// Calculate percent of register usage
IF ( CurrentAcrUsageCount > 0)
THEN
  CurrentAcrUsagePercent :=  (DINT_TO_REAL(CurrentAcrUsageCount) / DINT_TO_REAL(RegisterSize)) * 100.0;
ELSE
  CurrentAcrUsagePercent := 0.0;
END_IF

// build rising edge for arc usage over 80% 
WarningAcrUsage( CLK := CurrentAcrUsagePercent > RobotLibraryParameter.ACR_USAGE_WARNING_LIMIT );

IF ( WarningAcrUsage.Q )
THEN
  // Create log entry
  CreateLogMessagePara4( Timestamp   := SystemTime,
                         MessageType := MessageType.CMD,
                         Severity    := Severity.WARNING,
                         MessageCode := 0,
                         MessageText := 'ACR Register usage has reached the warning limit ({1}): {2}/{3} = {4}%',
                         Para1       :=  REAL_TO_STRING(RobotLibraryParameter.ACR_USAGE_WARNING_LIMIT),
                         Para2       :=  DINT_TO_STRING(CurrentAcrUsageCount),
                         Para3       :=  DINT_TO_STRING(RegisterSize),
                         Para4       :=  REAL_TO_STRING(CurrentAcrUsagePercent));  
END_IF
                
END_METHOD

METHOD PUBLIC OnOnlineChange : DINT
VAR_INPUT
  /// unique ID 
  UniqueID     : UDINT;
  /// Pointer to the corresponding command-FB to enable a callback mechanism
  pCommandFB   : POINTER TO RobotLibraryBaseFB;
END_VAR

VAR
  /// internal index for loops
 _regIdx : DINT;
END_VAR
                  OnOnlineChange := -1;

// Check command FB pointer is valid ?
IF ( pCommandFB <> RobotLibraryConstants.NULL_POINTER)
THEN
  FOR _regIdx := 1 TO RegisterSize
  DO
    // check unique ID found ?
    IF ( Register[_regIdx].UniqueID = UniqueID ) 
    THEN  
      // update pointer to command FB
      Register[_regIdx].pCommandFB := pCommandFB;
      // Return result OK
      OnOnlineChange := RobotLibraryConstants.OK;
      EXIT;
    END_IF
  END_FOR
END_IF
                
END_METHOD

METHOD PUBLIC RemoveCmd : DINT
VAR_INPUT
 /// unique ID
 UniqueID : UDINT;  
END_VAR

VAR
  /// internal index
 _regIdx : DINT;
  /// internal command type 
 _cmdType : CmdType;
END_VAR
                  RemoveCmd := RobotLibraryConstants.HAS_ERROR;


IF (UniqueID = 0)
THEN
  UniqueID := UniqueID;
END_IF

FOR _regIdx := 1 TO RegisterSize
DO
  // check unique ID found and not yet sended ?
  IF (( Register[_regIdx].UniqueID                  = UniqueID                        ) AND
      ( Register[_regIdx].Command[ACTIVE_CMD].State < BufferStateCmd.UPDATE_AVAILABLE ))       
  THEN
    // Get CmdType from payload
    SysDepMemCpy( pDest := ADR(_cmdType), pSrc := ADR(Register[_regIdx].Command[ACTIVE_CMD].Payload), DataLen := SIZEOF(_cmdType));
    // delete register entry
    SysDepMemSet(pDest := ADR(Register[_regIdx]), Value := 0 , DataLen := SIZEOF(Register[_regIdx]));
    // decrement current used register counter
    CurrentAcrUsageCount := CurrentAcrUsageCount - 1;
    // Command successfull removed
    RemoveCmd := RobotLibraryConstants.OK;    
    
    
    // Create log entry
    CreateLogMessagePara2 (  Timestamp   := SystemTime,
                             MessageType := MessageType.CMD,
                             Severity    := Severity.INFO,
                             MessageCode := 0,
                             MessageText := 'ACR-ID [{1}]: Removed CmdType <{2}>',
                             Para1       :=  DINT_TO_STRING(_regIdx),                 
                             Para2       :=  CMD_TYPE_TO_STRING(SwapUint(_cmdType)));
    EXIT;
  END_IF
END_FOR
                
END_METHOD

METHOD PUBLIC Reset
                  SysDepMemSet( ADR(Register), 0, SIZEOF(Register));              

CurrentAcrUsageCount   := 0;
CurrentAcrUsagePercent := 0.0;


// Create log entry
CreateLogMessagePara1 ( Timestamp   := SystemTime,
                        MessageType := MessageType.CMD,
                        Severity    := Severity.INFO,
                        MessageCode := 0,
                        MessageText := 'ACR Registers has been reset and all entries deleted by Reset method call',
                        Para1       :=  '');                          

                
END_METHOD

METHOD PRIVATE UpdateExecutionOrderList
VAR
  /// temporary Active Command Register entry
  TmpRegisterEntry : AxesGroupAcyclicAcrEntry;
  /// temporary index
  TmpIndex         : DINT;
  /// internal index
  i                : DINT;  
  /// internal index
  j                : DINT;  
END_VAR
                  // Reset temporary register
SysDepMemSet(pDest := ADR(TmpRegister)       , Value := 0, DataLen := SIZEOF(TmpRegister));
// Reset Execution Order List
SysDepMemSet(pDest := ADR(ExecutionOrderList), Value := 0, DataLen := SIZEOF(ExecutionOrderList));
// pre-set temporary register index 
j := 1;

FOR i := 1 TO RegisterSize
DO
  // add only entries which are not in status free and where datas must be processed
  IF (( Register[i].State                      > ActiveCommandRegisterState.IS_FREE ) AND
      ( Register[i].Command[ACTIVE_CMD].State <> BufferStateCmd.EMPTY               ) AND
      ( Register[i].Command[ACTIVE_CMD].State <> BufferStateCmd.PROCESSED           ))
  THEN
    // copy register entry 
    TmpRegister[j] := Register[i];
    // store index of the entry from the ACR
    ExecutionOrderList[j] := i;
    // inc temporar register index
    j := j + 1; 
  END_IF
END_FOR  

// Bubble Sort to sort the priorities from the active command register
FOR i := 1 TO RegisterSize
DO
  FOR j := 1 TO RegisterSize - 1
  DO 
    // check list entry is not empty ? 
    IF (( TmpRegister[i  ].State = ActiveCommandRegisterState.IS_FREE ) OR
        ( TmpRegister[j+1].State = ActiveCommandRegisterState.IS_FREE ))
    THEN
      EXIT; 
    END_IF  

    IF (( TmpRegister[j].Command[ACTIVE_CMD].Payload[PRIORITY_IDX] AND PRIORITY_BIT_MASK ) > ( TmpRegister[j+1].Command[ACTIVE_CMD].Payload[PRIORITY_IDX] AND PRIORITY_BIT_MASK ))
    THEN    
      // swap position of register entry  
      TmpRegisterEntry := TmpRegister[j];         
      TmpRegister[j]   := TmpRegister[j+1];
      TmpRegister[j+1] := TmpRegisterEntry;
      
      // swap position of index in the Execution Order List  
      TmpIndex                := ExecutionOrderList[j];
      ExecutionOrderList[j]   := ExecutionOrderList[j+1];
      ExecutionOrderList[j+1] := TmpIndex;
    END_IF
  END_FOR 
END_FOR

// Bubble Sort to sort the Timestamp from the pre-sorted active command register
FOR i := 1 TO RegisterSize
DO
  FOR j := 1 TO RegisterSize - 1
  DO    
    // check list entry is not empty ? 
    IF (( TmpRegister[i  ].State = ActiveCommandRegisterState.IS_FREE ) OR
        ( TmpRegister[j+1].State = ActiveCommandRegisterState.IS_FREE ))
    THEN
      EXIT; 
    END_IF  

       // Priority is higher
    IF (( TmpRegister[j].Command[ACTIVE_CMD].Payload[PRIORITY_IDX] AND PRIORITY_BIT_MASK ) >= ( TmpRegister[j+1].Command[ACTIVE_CMD].Payload[PRIORITY_IDX] AND PRIORITY_BIT_MASK )) AND
       // Date is greater 
       (( TmpRegister[j].Command[ACTIVE_CMD].Timestamp.SystemDate                          >    TmpRegister[j+1].Command[ACTIVE_CMD].Timestamp.SystemDate                         ) OR 
       // Date is the same, but Time is greater
       (( TmpRegister[j].Command[ACTIVE_CMD].Timestamp.SystemDate                          =    TmpRegister[j+1].Command[ACTIVE_CMD].Timestamp.SystemDate                         ) AND 
        ( TmpRegister[j].Command[ACTIVE_CMD].Timestamp.SystemTime                          >    TmpRegister[j+1].Command[ACTIVE_CMD].Timestamp.SystemTime                         )))
    THEN    
      // swap position of register entry  
      TmpRegisterEntry := TmpRegister[j];         
      TmpRegister[j]   := TmpRegister[j+1];
      TmpRegister[j+1] := TmpRegisterEntry;
      
      // swap position of index in the Execution Order List  
      TmpIndex                := ExecutionOrderList[j];
      ExecutionOrderList[j]   := ExecutionOrderList[j+1];
      ExecutionOrderList[j+1] := TmpIndex;
    END_IF
  END_FOR 
END_FOR
                
END_METHOD

PROPERTY PUBLIC NotifyParameterChanged : UDINT
SET
VAR
  /// internal register index
 _regIdx  : DINT;
  /// internal command type
 _cmdType : CmdType;
END_VAR
                    FOR _regIdx := 1 TO RobotLibraryParameter.ACTIVE_CMD_REGISTER_ENTRIES_MAX
DO
  // check unique ID found ?
  IF ( Register[_regIdx].UniqueID = NotifyParameterChanged )
  THEN  
    IF (( Register[_regIdx].Command[ACTIVE_CMD].State <> BufferStateCmd.SENDING   ) AND
        ( Register[_regIdx].Command[ACTIVE_CMD].State <> BufferStateCmd.PROCESSED ))
    THEN
      // Check pointer is valid ? 
      IF ( Register[_regIdx].pCommandFB <> RobotLibraryConstants.NULL_POINTER )
      THEN
        // add to send register
        Register[_regIdx].Command[ACTIVE_CMD].Timestamp  := SystemTime;
        Register[_regIdx].Command[ACTIVE_CMD].State      := BufferStateCmd.UPDATE_AVAILABLE;
        Register[_regIdx].Command[ACTIVE_CMD].Payload    := Register[_regIdx].pCommandFB^.CommandData.Payload;
        Register[_regIdx].Command[ACTIVE_CMD].PayloadLen := Register[_regIdx].pCommandFB^.CommandData.PayloadLen;

        // get command type from payload
       _cmdType := CombineBytesToUint(HiByte := Register[_regIdx].pCommandFB^.CommandData.Payload[0],
                                      LoByte := Register[_regIdx].pCommandFB^.CommandData.Payload[1]);
        
        // Create log entry
        CreateLogMessagePara2 ( Timestamp   := SystemTime,
                                MessageType := MessageType.CMD,
                                Severity    := Severity.INFO,
                                MessageCode := 0,
                                MessageText := 'ACR-ID [{1}]: Updated Cmd-Parameter of CmdType <{2}> -> written to ACTIVE_CMD Index',
                                Para1       :=  DINT_TO_STRING(_regIdx),
                                Para2       :=  CMD_TYPE_TO_STRING(_cmdType));
      END_IF
    ELSE
      // Check pointer is valid ? 
      IF ( Register[_regIdx].pCommandFB <> RobotLibraryConstants.NULL_POINTER )
      THEN
        // add to buffer register
        Register[_regIdx].Command[BUFFER_CMD].Timestamp  := SystemTime;
        Register[_regIdx].Command[BUFFER_CMD].State      := BufferStateCmd.UPDATE_AVAILABLE;
        Register[_regIdx].Command[BUFFER_CMD].Payload    := Register[_regIdx].pCommandFB^.CommandData.Payload;
        Register[_regIdx].Command[BUFFER_CMD].PayloadLen := Register[_regIdx].pCommandFB^.CommandData.PayloadLen;

        // get command type from payload
       _cmdType := CombineBytesToUint(HiByte := Register[_regIdx].pCommandFB^.CommandData.Payload[0],
                                      LoByte := Register[_regIdx].pCommandFB^.CommandData.Payload[1]);
        
        // Create log entry
        CreateLogMessagePara2 ( Timestamp   := SystemTime,
                                MessageType := MessageType.CMD,
                                Severity    := Severity.INFO,
                                MessageCode := 0,
                                MessageText := 'ACR-ID [{1}]: Updated Cmd-Parameter of CmdType <{2}> -> written to BUFFER_CMD Index',
                                Para1       :=  DINT_TO_STRING(_regIdx),
                                Para2       :=  CMD_TYPE_TO_STRING(_cmdType));
      END_IF
    END_IF
    
    
  END_IF
END_FOR
                  
END_SET
END_PROPERTY
END_FUNCTION_BLOCK

/// Abort triggering of Position, measuring input
FUNCTION_BLOCK MC_AbortMeasuringInputFB EXTENDS RobotLibraryBaseExecuteFB
// ------------------------------------------------------------------------- 
//  SRCI Robot Library                                                
// ------------------------------------------------------------------------- 
//                                                                           
//  Object:      AbortMeasuringInputFB                                       
//  Author:      Thorsten Brach                                                
//  Date:        2024-06-01
//
//  Description:                                              
//   
//                                                                           
//  Copyright: 
//    (C) 2024 Thorsten Brach. All rights reserved                                                                                                                                            
//             Licensed under the MIT License.
//                                                                           
//  Disclaimer:                                                                           
//    This project is provided without any guarantee and can be used for   
//    private and commercial purposes. Any use is at the user’s 
//    own risk and responsibility.
//
// -------------------------------------------------------------------------
VAR_INPUT
  /// Command parameter 
  ParCmd          : AbortMeasuringInputParCmd;      
END_VAR
VAR_OUTPUT
  /// Command is transferred and confirmed by the RC
  CommandBuffered : BOOL;  
  /// Command output 
  OutCmd          : AbortMeasuringInputOutCmd;          
END_VAR
VAR
  /// internal copy of command parameter 
 _parCmd          : AbortMeasuringInputParCmd;
  /// command data to send
 _command         : AbortMeasuringInputSendData;
  /// response data received
 _response        : AbortMeasuringInputRecvData;      
END_VAR

            SUPER^(AxesGroup := AxesGroup);
          

METHOD INTERNAL CheckAddParameter : BOOL
VAR_INPUT
  /// Payload pointer
  PayloadPtr : UDINT;
END_VAR
VAR
  /// Payload as byte array
  Payload    : ARRAY [1..SIZEOF(_command)] OF BYTE;
  /// Null Byte array 
  Null       : ARRAY [1..SIZEOF(_command)] OF BYTE;
  /// Data length to compare
  DataLen    : UDINT;
END_VAR
                  // Payload pointer must be decreased by one byte, because ADR(Payload) is already one byte !
PayloadPtr := LIMIT (0, PayloadPtr - 1, SIZEOF(Payload) -1);
// Convert command struct to payload array
SysDepMemCpy( pDest := ADR(Payload), pSrc := ADR(_command), DataLen := SIZEOF(_command));
// Calculate the data length to compare - at least one byte must be compared !
DataLen := LIMIT(1, SIZEOF(Payload) - PayloadPtr, SIZEOF(Payload)); 
// Compare Payload-Array with Null-Byte-Array
CheckAddParameter := SysDepMemCmp( pData1 := ADR(Payload) + PayloadPtr , pData2 := ADR(Null), DataLen := DataLen) <>  RobotLibraryConstants.OK ;
                
END_METHOD

METHOD PROTECTED CheckFunctionSupported : BOOL
VAR_IN_OUT
  /// Robot assignment of function
  AxesGroup : AxesGroup; 
END_VAR
                  CheckFunctionSupported := AxesGroup.State.RobotData.RCSupportedFunctions.AbortMeasuringInput;

IF ( NOT CheckFunctionSupported )
THEN
  // call base implementation for set error and create log entry
  SUPER^.CheckFunctionSupported(AxesGroup := AxesGroup);
END_IF
                
END_METHOD

METHOD PROTECTED CheckParameterChanged : BOOL
VAR_IN_OUT
  /// Robot assignment of function
  AxesGroup    : AxesGroup; 
END_VAR
                  // Check ParCmd Size is > 0, because MemCmp does not work correctly with size = 0
IF (SIZEOF(ParCmd) = 0) OR (_stepCmd = 0)
THEN 
  RETURN;
END_IF

// compare memory 
_parameterChanged := ( SysDepMemCmp(pData1 := ADR(ParCmd), pData2 := ADR(_parCmd), DataLen := SIZEOF(ParCmd)) <> RobotLibraryConstants.OK );

// check parameter valid ?
_parameterValid   := CheckParameterValid( AxesGroup := AxesGroup );

IF ((  _parameterChanged        )  AND 
    (  _parameterValid          )) OR
    (  _parameterUpdateInternal )  
THEN  
  // Create log entry for parameter changed event
  CreateLogMessagePara1 ( Timestamp   := AxesGroup.State.SystemTime,
                          MessageType := MessageType.CMD,
                          Severity    := Severity.DEBUG,
                          MessageCode := 0,
                          MessageText := 'NotifyParameterChanged Event {1}',
                          Para1       :=  '' );

  // reset internal flag for send parameter update
 _parameterUpdateInternal := FALSE;
  // update internal copy of parameters 
 _parCmd := ParCmd;
  // inc parameter sequence
 _command.ParSeq := _command.ParSeq + 1;
  // update command data  
  CommandData := CreateCommandPayload(AxesGroup := AxesGroup); // ( Access via reference to rCommandFB in ACR )
  // notify active command register 
  AxesGroup.Acyclic.ActiveCommandRegister.NotifyParameterChanged := _uniqueID;
END_IF
                
END_METHOD

METHOD PROTECTED CheckParameterValid : BOOL
VAR_IN_OUT
  /// Robot assignment of function
  AxesGroup : AxesGroup; 
END_VAR
                  CheckParameterValid := TRUE;


// Check ParCmd.MeasuringID valid ? 
IF ( ParCmd.MeasuringID < 0 )
THEN
  // Parameter not valid
  CheckParameterValid := FALSE;
  // Set error
  SetError( ErrorID := RobotLibraryErrorIdEnum.ERR_INVALID_PAR_CMD, Overwrite := TRUE ); 
  // Create log entry
  CreateLogMessagePara1 ( Timestamp   := AxesGroup.State.SystemTime,
                          MessageType := MessageType.CMD,
                          Severity    := Severity.ERROR,
                          MessageCode := ErrorID,
                          MessageText := 'Invalid Parameter ParCmd.MeasuringID = {1}',
                          Para1       := UINT_TO_STRING(ParCmd.MeasuringID));
  RETURN;                          
END_IF
                
END_METHOD

METHOD INTERNAL CreateCommandPayload : RobotLibraryCommandDataFB
VAR_IN_OUT
  /// Robot assignment of function
  AxesGroup : AxesGroup; 
END_VAR
VAR
  /// Parameter count
 _parameterCnt : DINT;
END_VAR
// Table 6-571: Sent CMD payload (PLC to RC) of "AbortMeasuringInput"
// --------------------------
// Header
// --------------------------
// Byte 000 : UINT  - Type HB     
// Byte 001 :       - Type LB    
// Byte 002 : USINT - Reserve | ExecutionMode
// Byte 003 : USINT - ParSeq  | Priority
// --------------------------
// Datablock
// --------------------------
// Byte 004 : UINT       - MeasuringID LW HB
// Byte 005 :            - MeasuringID LW LB
                  // set command parameter 
_command.CmdTyp      :=  CmdType.AbortMeasuringInput;
_command.ExecMode    :=  ExecMode;
_command.ParSeq      := _command.ParSeq;
_command.Priority    :=  Priority;
                     
_command.MeasuringID := parCmd.MeasuringID;

// copy command data to header
_cmdHeader := _command;
// call base implementation to copy header to payload buffer
CreateCommandPayload := SUPER^.CreateCommandPayload(AxesGroup := AxesGroup);


// Check parameter must be added ? 
IF ( CheckAddParameter(CreateCommandPayload.PayloadPtr))
THEN
  // add command.MeasuringID
  CreateCommandPayload.AddUint(_command.MeasuringID);
  // inc parameter counter
 _parameterCnt := _parameterCnt + 1;  
END_IF


// Create logging
CreateCommandPayloadLog(AxesGroup := AxesGroup, ParameterCnt := _parameterCnt);
                
END_METHOD

METHOD INTERNAL CreateCommandPayloadLog
VAR_IN_OUT
  /// Robot assignment of function
  AxesGroup : AxesGroup; 
END_VAR
VAR_INPUT
  /// Parameter count
  ParameterCnt : DINT;
END_VAR
                  // Create log entry for Parameter start
CreateLogMessagePara1 ( Timestamp   := AxesGroup.State.SystemTime,
                        MessageType := MessageType.CMD,
                        Severity    := Severity.DEBUG,
                        MessageCode := 0,
                        MessageText := 'Create command payload with {1} parameter(s) :',
                        Para1       := DINT_TO_STRING(ParameterCnt));
  

// Return if no parameter is remaining...
IF ( ParameterCnt = 0 ) THEN RETURN; END_IF
// dec remaining parameter(s)                        
ParameterCnt := ParameterCnt - 1;
// Create log entry for MeasuringID
CreateLogMessagePara1 ( Timestamp   := AxesGroup.State.SystemTime,
                        MessageType := MessageType.CMD,
                        Severity    := Severity.DEBUG,
                        MessageCode := 0,
                        MessageText := 'Command.MeasuringID = {1}',
                        Para1       :=  UINT_TO_STRING(_command.MeasuringID));

                
END_METHOD

METHOD FB_init : BOOL
VAR_INPUT
  /// if TRUE, the retain variables are initialized (warm start / cold start)
  bInitRetains : BOOL; 
  /// if TRUE, the instance afterwards gets moved into the copy code (online change)
  bInCopyCode  : BOOL;  
END_VAR
                  MyType := 'MC_AbortMeasuringInputFB';

ExecMode := ExecutionMode.PARALLEL;
Priority := PriorityLevel.NORMAL;
                
END_METHOD

METHOD PROTECTED OnExecRun : DINT
VAR_IN_OUT
  /// Robot assignment of function
  AxesGroup : AxesGroup; 
END_VAR
                  // call base implementation
SUPER^.OnExecRun(AxesGroup := AxesGroup);

CASE _stepCmd OF
  
  00:  IF ( _execute_R.Q ) AND ( NOT Error)
       THEN
         // Check function is supported and parameter are valid ?
         IF (( CheckFunctionSupported( AxesGroup := AxesGroup )) AND
             ( CheckParameterValid   ( AxesGroup := AxesGroup )))      
         THEN
           // set busy flag
           Busy := TRUE;
           // Reset command outputs
           SysDepMemSet(pDest := ADR(OutCmd), Value := 0, DataLen := SIZEOF(OutCmd));         
           // apply command parameter
          _parCmd := ParCmd;
           // init parameter sequence
          _command.ParSeq := 1;
           // create command data
           CommandData := CreateCommandPayload(AxesGroup := AxesGroup);
           // Add command to active command register
          _uniqueID := AxesGroup.Acyclic.ActiveCommandRegister.AddCmd( pCommandFB := ADR(THIS^ ));     
           // set timeout
           SetTimeout(PT := _timeoutCmd, rTimer := _timerCmd);
           // inc step counter
          _stepCmd := _stepCmd + 1;
         END_IF 
       END_IF


  01:  // Wait for responce received
       IF ( _responseReceived )
       THEN
         // reset response received flag
        _responseReceived := FALSE;
         // update state flags
         OnUpdateStateFlags(_response.State);
         // update state flags
         OnApplyOutCmd(_response.State);
                
         // Done, Aborted or Error ?
         IF (_response.State >= CmdMessageState.DONE )
         THEN
           // set timeout
           SetTimeout(PT := _timeoutCmd, rTimer := _timerCmd);
           // inc step counter
          _stepCmd := _stepCmd + 1; 
         END_IF
       END_IF


  02: IF ( NOT Execute)
      THEN
        Reset();
      END_IF     
ELSE
  // invalid step
  SetError( ErrorID := RobotLibraryErrorIdEnum.ERR_INVALID_STEP, Overwrite := TRUE );
END_CASE


// Reset FB
IF ( NOT Execute )
THEN
  Reset();
END_IF
                
END_METHOD

METHOD PROTECTED OnUpdateStateFlags
VAR_INPUT
  /// Command message state
  State : CmdMessageState;
END_VAR
                  // Reset State flags
Done:= FALSE;

CASE State OF

  // No operation or process is active
  CmdMessageState.EMPTY               :;
  // Created but not yet started
  CmdMessageState.CREATED             :;
  // Buffered and awaiting execution
  CmdMessageState.BUFFERED            : CommandBuffered := TRUE;
  // Buffered in planner for future execution
  CmdMessageState.BUFFERED_IN_PLANNER : CommandBuffered := TRUE;
  // Currently active and in progress
  CmdMessageState.ACTIVE              :;
  // Interrupted and awaiting continuation
  CmdMessageState.INTERRUPTED         :;
  // Requested for abort
  CmdMessageState.ABORT_REQUEST       :;
  // Successfully completed
  CmdMessageState.DONE                : Done  := TRUE;
                                        Busy  := FALSE;
  // Aborted before completion
  CmdMessageState.ABORTED             : Busy  := FALSE;
  // Encountered an error during execution
  CmdMessageState.ERROR               : Error := TRUE;
                                        Busy  := FALSE;
END_CASE
                
END_METHOD

METHOD INTERNAL ParseResponsePayload : DINT
VAR_INPUT
  /// Response data
  ResponseData : RobotLibraryResponseDataFB;
  /// Timestamp
  Timestamp    : SystemTime;  
END_VAR
VAR
  /// Parameter count
 _parameterCnt : DINT;
END_VAR
// Table 6-572: Received CMD payload (RC to PLC) of "AbortMeasuringInput"
// --------------------------
// Header
// --------------------------
// Byte 00 : USINT - ParSeq | State     
// Byte 01 : SINT  - AlarmMessageSeverity    
// Byte 02 : UINT  - AlarmMessageCode HB
// Byte 03 :       - AlarmMessageCode LB
                  // call base implementation to parse the header from payload buffer
ResponseData.PayloadPtr := SUPER^.ParseResponsePayload(ResponseData := ResponseData, Timestamp := Timestamp);

// copy parsed header to response
_response.ParSeq               := _rspHeader.ParSeq;
_response.State                := _rspHeader.State;
_response.AlarmMessageSeverity := _rspHeader.AlarmMessageSeverity;
_response.AlarmMessageCode     := _rspHeader.AlarmMessageCode;

// Create logging
ParseResponsePayloadLog(ResponseData := ResponseData, Timestamp := Timestamp, ParameterCnt := _parameterCnt);
                
END_METHOD

METHOD INTERNAL ParseResponsePayloadLog
VAR_INPUT
  /// Response data
  ResponseData : RobotLibraryResponseDataFB;
  /// Timestamp
  Timestamp    : SystemTime;  
  /// Parameter count
  ParameterCnt : DINT;
END_VAR
                  // Create log entry for Parameter start
CreateLogMessagePara1 ( Timestamp   := Timestamp,
                        MessageType := MessageType.CMD,
                        Severity    := Severity.DEBUG,
                        MessageCode := 0,
                        MessageText := '{1} parameter(s) to parse from the response data:',
                        Para1       := DINT_TO_STRING(ParameterCnt));
                        
// Return if no parameter is remaining...
IF ( ParameterCnt = 0 ) THEN RETURN; END_IF
// dec remaining parameter(s)                        
ParameterCnt := ParameterCnt - 1;
// Create log entry for no parameter 
CreateLogMessage      ( Timestamp   := Timestamp,
                        MessageType := MessageType.CMD,
                        Severity    := Severity.DEBUG,
                        MessageCode := 0,
                        MessageText := 'This command has no parameter to parse...');
                
END_METHOD

METHOD PROTECTED Reset : DINT
VAR_INPUT
END_VAR
                  Reset := SUPER^.Reset();

Done            := FALSE;
Busy            := FALSE;
CommandBuffered := FALSE;
                
END_METHOD
END_FUNCTION_BLOCK

/// Cancel currently active move command and continue with the next buffered command
FUNCTION_BLOCK MC_ActivateNextCommandFB EXTENDS RobotLibraryBaseExecuteFB
// ------------------------------------------------------------------------- 
//  SRCI Robot Library                                                
// ------------------------------------------------------------------------- 
//                                                                           
//  Object:      ActivateNextCommandFB                                       
//  Author:      Thorsten Brach                                                
//  Date:        2024-06-01
//
//  Description:                                              
//   
//                                                                           
//  Copyright: 
//    (C) 2024 Thorsten Brach. All rights reserved                                                                                                                                            
//             Licensed under the MIT License.
//                                                                           
//  Disclaimer:                                                                           
//    This project is provided without any guarantee and can be used for   
//    private and commercial purposes. Any use is at the user’s 
//    own risk and responsibility.
//
// -------------------------------------------------------------------------
VAR_INPUT
  /// Command parameter 
  ParCmd          : ActivateNextCommandParCmd;
  /// Processing mode
  ProcessingMode  : ProcessingMode;  
END_VAR
VAR_OUTPUT
  /// Command is transferred and confirmed by the RC
  CommandBuffered : BOOL;
  /// command results
  OutCmd          : ActivateNextCommandOutCmd;
END_VAR

VAR
  /// internal copy of command parameter 
 _parCmd          : ActivateNextCommandParCmd;
  /// command data to send
 _command         : ActivateNextCommandSendData;
  /// response data received
 _response        : ActivateNextCommandRecvData;   
  /// Trigger related EmitterID
 _emitterID       : ARRAY[0..3] OF SINT;
END_VAR

            SUPER^(AxesGroup := AxesGroup);
          

METHOD INTERNAL CheckAddParameter : BOOL
VAR_INPUT
  /// Payload pointer
  PayloadPtr : UDINT;
END_VAR
VAR
  /// Payload as byte array
  Payload    : ARRAY [1..SIZEOF(_command)] OF BYTE;
  /// Null Byte array 
  Null       : ARRAY [1..SIZEOF(_command)] OF BYTE;
  /// Data length to compare
  DataLen    : UDINT;
END_VAR
                  // Payload pointer must be decreased by one byte, because ADR(Payload) is already one byte !
PayloadPtr := LIMIT (0, PayloadPtr - 1, SIZEOF(Payload) -1);
// Convert command struct to payload array
SysDepMemCpy( pDest := ADR(Payload), pSrc := ADR(_command), DataLen := SIZEOF(_command));
// Calculate the data length to compare - at least one byte must be compared !
DataLen := LIMIT(1, SIZEOF(Payload) - PayloadPtr, SIZEOF(Payload)); 
// Compare Payload-Array with Null-Byte-Array
CheckAddParameter := SysDepMemCmp( pData1 := ADR(Payload) + PayloadPtr , pData2 := ADR(Null), DataLen := DataLen) <>  RobotLibraryConstants.OK ;
                
END_METHOD

METHOD PROTECTED CheckFunctionSupported : BOOL
VAR_IN_OUT
  /// Robot assignment of function
  AxesGroup : AxesGroup; 
END_VAR
                  CheckFunctionSupported := AxesGroup.State.RobotData.RCSupportedFunctions.ActivateNextCommand;

IF ( NOT CheckFunctionSupported )
THEN
  // call base implementation for set error and create log entry
  SUPER^.CheckFunctionSupported(AxesGroup := AxesGroup);
END_IF
                
END_METHOD

METHOD PROTECTED CheckParameterChanged : BOOL
VAR_IN_OUT
  /// Robot assignment of function
  AxesGroup    : AxesGroup; 
END_VAR
                  // Check ParCmd Size is > 0, because MemCmp does not work correctly with size = 0
IF (SIZEOF(ParCmd) = 0) OR (_stepCmd = 0)
THEN 
  RETURN;
END_IF

// compare memory 
_parameterChanged := ( SysDepMemCmp(pData1 := ADR(ParCmd), pData2 := ADR(_parCmd), DataLen := SIZEOF(ParCmd)) <> RobotLibraryConstants.OK );

// check parameter valid ?
_parameterValid   := CheckParameterValid( AxesGroup := AxesGroup );

IF ((  _parameterChanged        )  AND 
    (  _parameterValid          )) OR
    (  _parameterUpdateInternal )  
THEN  
  // Create log entry for parameter changed event
  CreateLogMessagePara1 ( Timestamp   := AxesGroup.State.SystemTime,
                          MessageType := MessageType.CMD,
                          Severity    := Severity.DEBUG,
                          MessageCode := 0,
                          MessageText := 'NotifyParameterChanged Event {1}',
                          Para1       :=  '' );

  // reset internal flag for send parameter update
 _parameterUpdateInternal := FALSE;
  // update internal copy of parameters 
 _parCmd := ParCmd;
  // inc parameter sequence
 _command.ParSeq := _command.ParSeq + 1;
  // update command data  
  CommandData := CreateCommandPayload(AxesGroup := AxesGroup); // ( Access via reference to rCommandFB in ACR )
  // notify active command register 
  AxesGroup.Acyclic.ActiveCommandRegister.NotifyParameterChanged := _uniqueID;  
END_IF
                
END_METHOD

METHOD PROTECTED CheckParameterValid : BOOL
VAR_IN_OUT
  /// Robot assignment of function
  AxesGroup : AxesGroup; 
END_VAR
                  CheckParameterValid := TRUE;

// Check ParCmd.ProcessingMode defined ? 
IF (( ProcessingMode < ProcessingModeEnum.BUFFERED         ) AND
    ( ProcessingMode > ProcessingModeEnum.TRIGGER_MULTIPLE ))
THEN
  // Parameter not valid
  CheckParameterValid := FALSE;
  // Set error
  SetError( ErrorID := RobotLibraryErrorIdEnum.ERR_PROCESSINGMODE_NOT_DEFINED, Overwrite := TRUE );
  // Create log entry
  CreateLogMessagePara1 ( Timestamp   := AxesGroup.State.SystemTime,
                          MessageType := MessageType.CMD,
                          Severity    := Severity.ERROR,
                          MessageCode := ErrorID,
                          MessageText := 'Invalid Parameter ParCmd.ProcessingMode = {1}',
                          Para1       := PROCESSING_MODE_TO_STRING(ProcessingMode));
  RETURN;                          
END_IF


// Check ParCmd.ProcessingMode valid ? 
IF (( ProcessingMode <> ProcessingModeEnum.PARALLEL         ) AND
    ( ProcessingMode <> ProcessingModeEnum.DEACTIVATE       ) AND
    ( ProcessingMode <> ProcessingModeEnum.TRIGGER_ONCE     ) AND
    ( ProcessingMode <> ProcessingModeEnum.TRIGGER_MULTIPLE ))
THEN
  // Parameter not valid
  CheckParameterValid := FALSE;
  // Set error
  SetError( ErrorID := RobotLibraryErrorIdEnum.ERR_PROCESSINGMODE_NOT_ALLOWED, Overwrite := TRUE );
  // Create log entry
  CreateLogMessagePara1 ( Timestamp   := AxesGroup.State.SystemTime,
                          MessageType := MessageType.CMD,
                          Severity    := Severity.ERROR,
                          MessageCode := ErrorID,
                          MessageText := 'Invalid Parameter ParCmd.ProcessingMode = {1}',
                          Para1       := PROCESSING_MODE_TO_STRING(ProcessingMode));
  RETURN;                          
END_IF


// Check ParCmd.ListenerID valid ? 
IF (( ParCmd.ListenerID <   0 ) OR 
    ( ParCmd.ListenerID > 127 ))
THEN
  // Parameter not valid
  CheckParameterValid := FALSE;
  // Set error
  SetError( ErrorID := RobotLibraryErrorIdEnum.ERR_LISTENERID_MUST_BE_POSITIVE, Overwrite := TRUE );
  // Create log entry
  CreateLogMessagePara1 ( Timestamp   := AxesGroup.State.SystemTime,
                          MessageType := MessageType.CMD,
                          Severity    := Severity.ERROR,
                          MessageCode := ErrorID,
                          MessageText := 'Invalid Parameter ParCmd.ListenerID = {1}',
                          Para1       := SINT_TO_STRING(ParCmd.ListenerID));                            
  RETURN;
END_IF


                
END_METHOD

METHOD INTERNAL CreateCommandPayload : RobotLibraryCommandDataFB
VAR_IN_OUT
  /// Robot assignment of function
  AxesGroup : AxesGroup; 
END_VAR
VAR
  /// Parameter count
 _parameterCnt : DINT;
END_VAR
// Table 6-662: Sent CMD payload (PLC to RC) of "ActivateNextCommand"
// --------------------------
// Header
// --------------------------
// Byte 00 : UINT  - Type HB     
// Byte 01 :       - Type LB    
// Byte 02 : USINT - Reserve | ExecutionMode
// Byte 03 : USINT - ParSeq  | Priority
// --------------------------
// Datablock
// --------------------------
// Byte 04 : SINT - EmitterID[0]
// Byte 05 : SINT - EmitterID[1]
// Byte 06 : SINT - EmitterID[2]   
// Byte 07 : SINT - EmitterID[3]
// Byte 08 : SINT - ListenerID
// Byte 09 : BYTE - Reserve
// --------------------------
                  // set command parameter 
_command.CmdTyp     :=  CmdType.ActivateNextCommand;
_command.ExecMode   :=  ExecMode;
_command.ParSeq     := _command.ParSeq;
_command.Priority   :=  Priority;
_command.ListenerID := _parCmd.ListenerID;


// copy command data to header
_cmdHeader := _command;
// call base implementation to copy header to payload buffer
CreateCommandPayload := SUPER^.CreateCommandPayload(AxesGroup := AxesGroup);


// Check parameter must be added ? 
IF ( CheckAddParameter(CreateCommandPayload.PayloadPtr))
THEN
  // add command.EmitterID[0]
  CreateCommandPayload.AddSint(_command.EmitterID[0]);
  // inc parameter counter
 _parameterCnt := _parameterCnt + 1;  
END_IF


// Check parameter must be added ? 
IF ( CheckAddParameter(CreateCommandPayload.PayloadPtr))
THEN
  // add command.EmitterID[1]
  CreateCommandPayload.AddSint(_command.EmitterID[1]);
  // inc parameter counter
 _parameterCnt := _parameterCnt + 1;  
END_IF


// Check parameter must be added ? 
IF ( CheckAddParameter(CreateCommandPayload.PayloadPtr))
THEN
  // add command.EmitterID[2]
  CreateCommandPayload.AddSint(_command.EmitterID[2]);
  // inc parameter counter
 _parameterCnt := _parameterCnt + 1;  
END_IF


// Check parameter must be added ? 
IF ( CheckAddParameter(CreateCommandPayload.PayloadPtr))
THEN
  // add command.EmitterID[3]
  CreateCommandPayload.AddSint(_command.EmitterID[3]);
  // inc parameter counter
 _parameterCnt := _parameterCnt + 1;  
END_IF


// Check parameter must be added ? 
IF ( CheckAddParameter(CreateCommandPayload.PayloadPtr))
THEN
  // add command.ListenerID
  CreateCommandPayload.AddSint(_command.ListenerID);
  // inc parameter counter
 _parameterCnt := _parameterCnt + 1;  
END_IF


// Check parameter must be added ? 
IF ( CheckAddParameter(CreateCommandPayload.PayloadPtr))
THEN
  // add command.Reserve
  CreateCommandPayload.AddByte(_command.Reserve);
  // inc parameter counter
 _parameterCnt := _parameterCnt + 1;  
END_IF
  
  
// Create logging
CreateCommandPayloadLog(AxesGroup := AxesGroup, ParameterCnt := _parameterCnt);
                
END_METHOD

METHOD INTERNAL CreateCommandPayloadLog
VAR_IN_OUT
  /// Robot assignment of function
  AxesGroup : AxesGroup; 
END_VAR
VAR_INPUT
  /// Parameter count
  ParameterCnt : DINT;
END_VAR
VAR 
  /// internal index for loops
 _idx : DINT;
END_VAR
                  // Create log entry for Parameter start
CreateLogMessagePara1 ( Timestamp   := AxesGroup.State.SystemTime,
                        MessageType := MessageType.CMD,
                        Severity    := Severity.DEBUG,
                        MessageCode := 0,
                        MessageText := 'Create command payload with {1} parameter(s) :',
                        Para1       := DINT_TO_STRING(ParameterCnt));
  
// Create log entry for EmitterID[x]
FOR _idx := 0 TO 3
DO
  // Return if no parameter is remaining...
  IF ( ParameterCnt = 0 ) THEN RETURN; END_IF
  // dec remaining parameter(s)                        
  ParameterCnt := ParameterCnt - 1;
  // Create log entry for Command.EmitterID
  CreateLogMessagePara2 ( Timestamp   := AxesGroup.State.SystemTime,
                          MessageType := MessageType.CMD,
                          Severity    := Severity.DEBUG,
                          MessageCode := 0,
                          MessageText := 'Command.EmitterID[{2}] = {1}',
                          Para1       :=  SINT_TO_STRING(_command.EmitterID[_idx]),
                          Para2       :=  DINT_TO_STRING(_idx));
END_FOR


// Return if no parameter is remaining...
IF ( ParameterCnt = 0 ) THEN RETURN; END_IF
// dec remaining parameter(s)                        
ParameterCnt := ParameterCnt - 1;
// Create log entry for ListenerID
CreateLogMessagePara1 ( Timestamp   := AxesGroup.State.SystemTime,
                        MessageType := MessageType.CMD,
                        Severity    := Severity.DEBUG,
                        MessageCode := 0,
                        MessageText := 'Command.ListenerID = {1}',
                        Para1       :=  SINT_TO_STRING(_command.ListenerID));


// Return if no parameter is remaining...
IF ( ParameterCnt = 0 ) THEN RETURN; END_IF
// dec remaining parameter(s)                        
ParameterCnt := ParameterCnt - 1;
// Create log entry for Reserve
CreateLogMessagePara1 ( Timestamp   := AxesGroup.State.SystemTime,
                        MessageType := MessageType.CMD,
                        Severity    := Severity.DEBUG,
                        MessageCode := 0,
                        MessageText := 'Command.Reserve = {1}',
                        Para1       :=  BYTE_TO_STRING(_command.Reserve));
                
END_METHOD

METHOD FB_init : BOOL
VAR_INPUT
  /// if TRUE, the retain variables are initialized (warm start / cold start)
  bInitRetains : BOOL; 
  /// if TRUE, the instance afterwards gets moved into the copy code (online change)
  bInCopyCode  : BOOL;  
END_VAR
                  MyType := 'MC_ActivateNextCommandFB';

ExecMode       := ExecutionMode.PARALLEL;
Priority       := PriorityLevel.NORMAL;
ProcessingMode := ProcessingModeEnum.PARALLEL;
                
END_METHOD

METHOD PROTECTED OnApplyOutCmd
VAR_INPUT
  /// Command message state
  State : CmdMessageState;
END_VAR
                  IF ( State = CmdMessageState.EMPTY ) 
THEN
  // Reset command outputs
  SysDepMemSet(pDest := ADR(OutCmd), Value := 0, DataLen := SIZEOF(OutCmd));         
END_IF

IF ( State = CmdMessageState.DONE ) 
THEN
  OutCmd.InvocationCounter := _response.InvocationCounter;
  OutCmd.OriginID          := _response.OriginID;
END_IF
                
END_METHOD

METHOD PROTECTED OnExecRun : DINT
VAR_IN_OUT
  /// Robot assignment of function
  AxesGroup : AxesGroup; 
END_VAR
                  // call base implementation
SUPER^.OnExecRun(AxesGroup := AxesGroup);

CASE _stepCmd OF
  
  00:  IF ( _execute_R.Q ) AND ( NOT Error) 
       THEN
         // Check function is supported and parameter are valid ?
         IF (( CheckFunctionSupported( AxesGroup := AxesGroup )) AND
             ( CheckParameterValid   ( AxesGroup := AxesGroup )))      
         THEN
           // set busy flag
           Busy := TRUE;
           // Reset command outputs
           SysDepMemSet(pDest := ADR(OutCmd), Value := 0, DataLen := SIZEOF(OutCmd));         
           // apply command parameter
          _parCmd := ParCmd;
           // init parameter sequence
          _command.ParSeq := 1;
           // create command data
           CommandData := CreateCommandPayload(AxesGroup := AxesGroup);
           // Add command to active command register
          _uniqueID := AxesGroup.Acyclic.ActiveCommandRegister.AddCmd( pCommandFB := ADR(THIS^ ));     
           // set timeout
           SetTimeout(PT := _timeoutCmd, rTimer := _timerCmd);
           // inc step counter
          _stepCmd := _stepCmd + 1;
         END_IF 
       END_IF


  01:  // Wait for responce received
       IF ( _responseReceived )
       THEN
         // reset response received flag
        _responseReceived := FALSE;
         // update state flags
         OnUpdateStateFlags(_response.State);
         // update state flags
         OnApplyOutCmd(_response.State);

         // Done, Aborted or Error ?
         IF (_response.State >= CmdMessageState.DONE )
         THEN
           // set timeout
           SetTimeout(PT := _timeoutCmd, rTimer := _timerCmd);
           // inc step counter
          _stepCmd := _stepCmd + 1; 
         END_IF
       END_IF


  02: IF ( NOT Execute)
      THEN
        Reset();
       END_IF     
ELSE
  // invalid step
  SetError( ErrorID := RobotLibraryErrorIdEnum.ERR_INVALID_STEP, Overwrite := TRUE );
END_CASE


// Reset FB
IF ( NOT Execute )
THEN
  Reset();  
END_IF
                
END_METHOD

METHOD PROTECTED OnUpdateStateFlags
VAR_INPUT
  /// Command message state
  State : CmdMessageState;
END_VAR
                  // Reset State flags
Done := FALSE;

CASE State OF

  // No operation or process is active
  CmdMessageState.EMPTY               :;
  // Created but not yet started
  CmdMessageState.CREATED             :;
  // Buffered and awaiting execution
  CmdMessageState.BUFFERED            : CommandBuffered := TRUE;
  // Buffered in planner for future execution
  CmdMessageState.BUFFERED_IN_PLANNER : CommandBuffered := TRUE;
  // Currently active and in progress
  CmdMessageState.ACTIVE              :;
  // Interrupted and awaiting continuation
  CmdMessageState.INTERRUPTED         :;
  // Requested for abort
  CmdMessageState.ABORT_REQUEST       :;
  // Successfully completed
  CmdMessageState.DONE                : Done := TRUE;
                                        Busy := FALSE;
  // Aborted before completion
  CmdMessageState.ABORTED             : Busy := FALSE;
  // Encountered an error during execution
  CmdMessageState.ERROR               : Busy := FALSE;
END_CASE
                
END_METHOD

METHOD INTERNAL ParseResponsePayload : DINT
VAR_INPUT
  /// Response data
  ResponseData : RobotLibraryResponseDataFB;
  /// Timestamp
  Timestamp    : SystemTime;  
END_VAR
VAR
  /// Parameter count
 _parameterCnt : DINT;
END_VAR
// Table 6-663: Received CMD payload (RC to PLC) of "ActivateNextCommand"
// --------------------------
// Header
// --------------------------
// Byte 00 : USINT - ParSeq | State     
// Byte 01 : SINT  - AlarmMessageSeverity    
// Byte 02 : UINT  - AlarmMessageCode HB
// Byte 03 :       - AlarmMessageCode LB
// --------------------------
// Datablock
// --------------------------
// Byte 04 : USINT - InvocationCounter
// Byte 05 : SINT  - Reserved
// Byte 06 : INT   - OriginID HB
// Byte 07 : INT   - OriginID LB
// --------------------------
                  // call base implementation to parse the header from payload buffer
ResponseData.PayloadPtr := SUPER^.ParseResponsePayload(ResponseData := ResponseData, Timestamp := Timestamp);

// copy parsed header to response
_response.ParSeq               := _rspHeader.ParSeq;
_response.State                := _rspHeader.State;
_response.AlarmMessageSeverity := _rspHeader.AlarmMessageSeverity;
_response.AlarmMessageCode     := _rspHeader.AlarmMessageCode;


// Check payload remaining ? 
IF ( ResponseData.IsPayloadRemaining)
THEN
  // Get InvocationCounter
 _response.InvocationCounter := ResponseData.GetUsint();
  // inc parameter counter
 _parameterCnt := _parameterCnt + 1;
END_IF


// Check payload remaining ? 
IF ( ResponseData.IsPayloadRemaining)
THEN
  // Get Reserve
 _response.Reserve := ResponseData.GetSint();
  // inc parameter counter
 _parameterCnt := _parameterCnt + 1;
END_IF


// Check payload remaining ? 
IF ( ResponseData.IsPayloadRemaining)
THEN
  // Get OriginID
 _response.OriginID := ResponseData.GetInt();
  // inc parameter counter
 _parameterCnt := _parameterCnt + 1;
END_IF


// Create logging
ParseResponsePayloadLog(ResponseData := ResponseData, Timestamp := Timestamp, ParameterCnt := _parameterCnt);
                
END_METHOD

METHOD INTERNAL ParseResponsePayloadLog
VAR_INPUT
  /// Response data
  ResponseData : RobotLibraryResponseDataFB;
  /// Timestamp
  Timestamp    : SystemTime;  
  /// Parameter count
  ParameterCnt : DINT;  
END_VAR
                  // Create log entry for Parameter start
CreateLogMessagePara1 ( Timestamp   := Timestamp,
                        MessageType := MessageType.CMD,
                        Severity    := Severity.DEBUG,
                        MessageCode := 0,
                        MessageText := '{1} parameter(s) to parse from the response data:',
                        Para1       := DINT_TO_STRING(ParameterCnt));

                        
// Return if no parameter is remaining...
IF ( ParameterCnt = 0 ) THEN RETURN; END_IF
// dec remaining parameter(s)                        
ParameterCnt := ParameterCnt - 1;
// Create log entry for InvocationCounter
CreateLogMessagePara1 ( Timestamp   := Timestamp,
                        MessageType := MessageType.CMD,
                        Severity    := Severity.DEBUG,
                        MessageCode := 0,
                        MessageText := 'Response.InvocationCounter = {1}',
                        Para1       :=  USINT_TO_STRING(_response.InvocationCounter));


// Return if no parameter is remaining...
IF ( ParameterCnt = 0 ) THEN RETURN; END_IF
// dec remaining parameter(s)                        
ParameterCnt := ParameterCnt - 1;
// Create log entry for Reserve
CreateLogMessagePara1 ( Timestamp   := Timestamp,
                        MessageType := MessageType.CMD,
                        Severity    := Severity.DEBUG,
                        MessageCode := 0,
                        MessageText := 'Response.Reserve = {1}',
                        Para1       :=  SINT_TO_STRING(_response.Reserve));


// Return if no parameter is remaining...
IF ( ParameterCnt = 0 ) THEN RETURN; END_IF
// dec remaining parameter(s)                        
ParameterCnt := ParameterCnt - 1;
// Create log entry for OriginID
CreateLogMessagePara1 ( Timestamp   := Timestamp,
                        MessageType := MessageType.CMD,
                        Severity    := Severity.DEBUG,
                        MessageCode := 0,
                        MessageText := 'Response.OriginID = {1}',
                        Para1       :=  INT_TO_STRING(_response.OriginID));
                
END_METHOD

METHOD PROTECTED Reset : DINT
VAR_INPUT
END_VAR
                  Reset := SUPER^.Reset();

Done            := FALSE;
Busy            := FALSE;
CommandBuffered := FALSE;
                
END_METHOD
END_FUNCTION_BLOCK

/// Activate/Deactivate functionality to avoid singularities
FUNCTION_BLOCK MC_AvoidSingularityFB EXTENDS RobotLibraryBaseEnableFB
// ------------------------------------------------------------------------- 
//  SRCI Robot Library                                                
// ------------------------------------------------------------------------- 
//                                                                           
//  Object:      AvoidSingularityFB                                       
//  Author:      Thorsten Brach                                                
//  Date:        2024-06-01
//
//  Description:                                              
//   
//                                                                           
//  Copyright: 
//    (C) 2024 Thorsten Brach. All rights reserved                                                                                                                                            
//             Licensed under the MIT License.
//                                                                           
//  Disclaimer:                                                                           
//    This project is provided without any guarantee and can be used for   
//    private and commercial purposes. Any use is at the user’s 
//    own risk and responsibility.
//
// -------------------------------------------------------------------------
VAR_INPUT
  /// Command parameter 
  ParCmd            : AvoidSingularityParCmd;
END_VAR

VAR_OUTPUT
  /// Command is transferred and confirmed by the RC
  CommandBuffered   : BOOL;
  /// Receiving of input parameter values has been acknowledged by RC
  ParameterAccepted : BOOL;
  /// command results
  OutCmd            : AvoidSingularityOutCmd;  
END_VAR


VAR
  /// internal copy of command parameter 
 _parCmd            : AvoidSingularityParCmd;
  /// command data to send
 _command           : AvoidSingularitySendData;
  /// response data received
 _response          : AvoidSingularityRecvData;
END_VAR

            SUPER^(AxesGroup := AxesGroup);
          

METHOD INTERNAL CheckAddParameter : BOOL
VAR_INPUT
  /// Payload pointer
  PayloadPtr : UDINT;
END_VAR
VAR
  /// Payload as byte array
  Payload    : ARRAY [1..SIZEOF(_command)] OF BYTE;
  /// Null Byte array 
  Null       : ARRAY [1..SIZEOF(_command)] OF BYTE;
  /// Data length to compare
  DataLen    : UDINT;
END_VAR
                  // Payload pointer must be decreased by one byte, because ADR(Payload) is already one byte !
PayloadPtr := LIMIT (0, PayloadPtr - 1, SIZEOF(Payload) -1);
// Convert command struct to payload array
SysDepMemCpy( pDest := ADR(Payload), pSrc := ADR(_command), DataLen := SIZEOF(_command));
// Calculate the data length to compare - at least one byte must be compared !
DataLen := LIMIT(1, SIZEOF(Payload) - PayloadPtr, SIZEOF(Payload)); 
// Compare Payload-Array with Null-Byte-Array
CheckAddParameter := SysDepMemCmp( pData1 := ADR(Payload) + PayloadPtr , pData2 := ADR(Null), DataLen := DataLen) <>  RobotLibraryConstants.OK ;
                
END_METHOD

METHOD PROTECTED CheckFunctionSupported : BOOL
VAR_IN_OUT
  /// Robot assignment of function
  AxesGroup : AxesGroup; 
END_VAR
                  CheckFunctionSupported := AxesGroup.State.RobotData.RCSupportedFunctions.AvoidSingularity;

IF ( NOT CheckFunctionSupported )
THEN
  // call base implementation for set error and create log entry
  SUPER^.CheckFunctionSupported(AxesGroup := AxesGroup);
END_IF
                
END_METHOD

METHOD PROTECTED CheckParameterChanged : BOOL
VAR_IN_OUT
  /// Robot assignment of function
  AxesGroup    : AxesGroup; 
END_VAR
                  // Check ParCmd Size is > 0, because MemCmp does not work correctly with size = 0
IF (SIZEOF(ParCmd) = 0) OR (_stepCmd = 0)
THEN 
  RETURN;
END_IF

// compare memory 
_parameterChanged := ( SysDepMemCmp(pData1 := ADR(ParCmd), pData2 := ADR(_parCmd), DataLen := SIZEOF(ParCmd)) <> RobotLibraryConstants.OK );

// check parameter valid ?
_parameterValid   := CheckParameterValid( AxesGroup := AxesGroup );

IF ((  _parameterChanged        )  AND 
    (  _parameterValid          )) OR
    (  _parameterUpdateInternal )  
THEN  
  // Create log entry for parameter changed event
  CreateLogMessagePara1 ( Timestamp   := AxesGroup.State.SystemTime,
                          MessageType := MessageType.CMD,
                          Severity    := Severity.DEBUG,
                          MessageCode := 0,
                          MessageText := 'NotifyParameterChanged Event {1}',
                          Para1       :=  '' );

  // reset internal flag for send parameter update
 _parameterUpdateInternal := FALSE;
  // update internal copy of parameters 
 _parCmd := ParCmd;
  // inc parameter sequence
 _command.ParSeq := _command.ParSeq + 1;
  // update command data  
  CommandData := CreateCommandPayload(AxesGroup := AxesGroup); // ( Access via reference to rCommandFB in ACR )
  // notify active command register 
  AxesGroup.Acyclic.ActiveCommandRegister.NotifyParameterChanged := _uniqueID;  
  // Reset parameter accepted flag
  ParameterAccepted := FALSE;
END_IF
                
END_METHOD

METHOD PROTECTED CheckParameterValid : BOOL
VAR_IN_OUT
  /// Robot assignment of function
  AxesGroup : AxesGroup; 
END_VAR
                  CheckParameterValid := TRUE;

// Check ParCmd.Mode valid ? 
IF (( ParCmd.Mode <> SingularityAvoidanceMode.NO_CHANGE        ) AND  
    ( ParCmd.Mode <> SingularityAvoidanceMode.LOCK_J4          ) AND
    ( ParCmd.Mode <> SingularityAvoidanceMode.TOOL_ORIENTATION ))
THEN
  // Parameter not valid
  CheckParameterValid := FALSE;
  // Set error
  SetError( ErrorID := RobotLibraryErrorIdEnum.ERR_INVALID_PAR_CMD, Overwrite := TRUE ); 
  // Create log entry
  CreateLogMessagePara1 ( Timestamp   := AxesGroup.State.SystemTime,
                          MessageType := MessageType.CMD,
                          Severity    := Severity.ERROR,
                          MessageCode := ErrorID,
                          MessageText := 'Invalid Parameter ParCmd.Mode = {1}',
                          Para1       := SINGULARITY_AVOIDANCE_MODE_TO_STRING(ParCmd.Mode));
  RETURN;                          
END_IF
                
END_METHOD

METHOD INTERNAL CreateCommandPayload : RobotLibraryCommandDataFB
VAR_IN_OUT
  /// Robot assignment of function
  AxesGroup : AxesGroup; 
END_VAR
VAR
  /// Parameter count
 _parameterCnt : DINT;
END_VAR
// Table 6-709: Sent CMD payload (PLC to RC) of "AvoidSingularity"
// --------------------------
// Header
// --------------------------
// Byte 00 : UINT  - Type HB     
// Byte 01 :       - Type LB    
// Byte 02 : USINT - Reserve | ExecutionMode
// Byte 03 : USINT - ParSeq  | Priority
// --------------------------
// Datablock
// --------------------------
// Byte 04 : BOOL   - Enable
// Byte 05 : USINT  - Mode
// --------------------------
                  // set command parameter 
_command.CmdTyp    :=  CmdType.AvoidSingularity;
_command.ExecMode  :=  ExecMode;
_command.ParSeq    := _command.ParSeq;
_command.Priority  :=  Priority;
_command.Enable    :=  Enable;
_command.Mode      := _parCmd.Mode;

// copy command data to header
_cmdHeader := _command;
// call base implementation to copy header to payload buffer
CreateCommandPayload := SUPER^.CreateCommandPayload(AxesGroup := AxesGroup);


// Check parameter must be added ? 
IF ( CheckAddParameter(CreateCommandPayload.PayloadPtr))
THEN
  // add command.Enable
  CreateCommandPayload.AddBool(_command.Enable);
  // inc parameter counter
 _parameterCnt := _parameterCnt + 1;  
END_IF


// Check parameter must be added ? 
IF ( CheckAddParameter(CreateCommandPayload.PayloadPtr))
THEN
  // add command.Mode
  CreateCommandPayload.AddByte(_command.Mode);
  // inc parameter counter
 _parameterCnt := _parameterCnt + 1;  
END_IF


// Create logging
CreateCommandPayloadLog(AxesGroup := AxesGroup, ParameterCnt := _parameterCnt);
                
END_METHOD

METHOD INTERNAL CreateCommandPayloadLog
VAR_IN_OUT
  /// Robot assignment of function
  AxesGroup : AxesGroup; 
END_VAR
VAR_INPUT
  /// Parameter count
  ParameterCnt : DINT;
END_VAR
                  // Create log entry for Parameter start
CreateLogMessagePara1 ( Timestamp   := AxesGroup.State.SystemTime,
                        MessageType := MessageType.CMD,
                        Severity    := Severity.DEBUG,
                        MessageCode := 0,
                        MessageText := 'Create command payload with {1} parameter(s) :',
                        Para1       := DINT_TO_STRING(ParameterCnt));
  

// Return if no parameter is remaining...
IF ( ParameterCnt = 0 ) THEN RETURN; END_IF
// dec remaining parameter(s)                        
ParameterCnt := ParameterCnt - 1;
// Create log entry for Enable
CreateLogMessagePara1 ( Timestamp   := AxesGroup.State.SystemTime,
                        MessageType := MessageType.CMD,
                        Severity    := Severity.DEBUG,
                        MessageCode := 0,
                        MessageText := 'Command.Enable = {1}',
                        Para1       :=  BOOL_TO_STRING(_command.Enable));


// Return if no parameter is remaining...
IF ( ParameterCnt = 0 ) THEN RETURN; END_IF
// dec remaining parameter(s)                        
ParameterCnt := ParameterCnt - 1;
// Create log entry for Mode
CreateLogMessagePara1 ( Timestamp   := AxesGroup.State.SystemTime,
                        MessageType := MessageType.CMD,
                        Severity    := Severity.DEBUG,
                        MessageCode := 0,
                        MessageText := 'Command.Mode = {1}',
                        Para1       :=  SINGULARITY_AVOIDANCE_MODE_TO_STRING(_command.Mode));

                
END_METHOD

METHOD FB_init : BOOL
VAR_INPUT
  /// if TRUE, the retain variables are initialized (warm start / cold start)
  bInitRetains : BOOL; 
  /// if TRUE, the instance afterwards gets moved into the copy code (online change)
  bInCopyCode  : BOOL;  
END_VAR
                  MyType := 'MC_AvoidSingularityFB';

ExecMode := ExecutionMode.PARALLEL;
Priority := PriorityLevel.NORMAL;
                
END_METHOD

METHOD Protected OnExecCancel : DINT
VAR_IN_OUT
  /// Robot assignment of function
  AxesGroup : AxesGroup; 
END_VAR
VAR
  /// internal return value 
 _retVal    : DINT;
END_VAR
                  OnExecCancel := RobotLibraryConstants.RUNNING;

CASE _stepCancel OF
  
  0: // set busy flag
     Busy := TRUE;
    
     // Create log entry
     CreateLogMessagePara1 ( Timestamp   := AxesGroup.State.SystemTime,
                             MessageType := MessageType.CMD,
                             Severity    := Severity.DEBUG,
                             MessageCode := 0,
                             MessageText := 'Execution of {1} cancelled',
                             Para1       := MyType);                 
    
     // try to remove cmd
    _retVal := AxesGroup.Acyclic.ActiveCommandRegister.RemoveCmd(_uniqueID);
  
     // check result of removement       
     IF ( _retVal = RobotLibraryConstants.OK )
     THEN
       // Reset step counter
      _stepCancel := 0;
       // finished okay
       OnExecCancel := RobotLibraryConstants.OK;
     
       // Create log entry
       CreateLogMessagePara1 ( Timestamp   := AxesGroup.State.SystemTime,
                               MessageType := MessageType.CMD,
                               Severity    := Severity.DEBUG,
                               MessageCode := 0,
                               MessageText := '{1} successfully removed from ACR',
                               Para1       := MyType);                 
     ELSE
       // set timeout
       SetTimeout(PT := _timeoutCancel, rTimer := _timerCancel);
       // inc step counter
      _stepCancel := _stepCancel + 1; 
     
       // Create log entry
       CreateLogMessagePara1 ( Timestamp   := AxesGroup.State.SystemTime,
                               MessageType := MessageType.CMD,
                               Severity    := Severity.DEBUG,
                               MessageCode := 0,
                               MessageText := '{1} was not removed from ACR because execution was already in progress',
                               Para1       := MyType);                 
     END_IF       
  
     
 1:  // call clear error 
     OnExecCancel := OnExecErrorClear(AxesGroup := AxesGroup);  
 
     IF ( OnExecCancel = RobotLibraryConstants.OK)
     THEN
       // Reset busy flag
       Busy := FALSE;
       // Reset step counter
      _stepCancel := 0;
       // finished okay
       OnExecCancel := RobotLibraryConstants.OK;
     END_IF  
  
ELSE
  // invalid step
  SetError( ErrorID := RobotLibraryErrorIdEnum.ERR_INVALID_STEP, Overwrite := TRUE );
END_CASE  


                        
// reset step counter
IF (OnExecCancel <> RobotLibraryConstants.RUNNING)
THEN
  // Reset FB variables
  Reset();
  // Reset step counter
 _stepCancel := 0;
END_IF                        
                
END_METHOD

METHOD PROTECTED OnExecErrorClear : DINT
VAR_IN_OUT
  /// Robot assignment of function
  AxesGroup : AxesGroup; 
END_VAR
                  OnExecErrorClear := RobotLibraryConstants.RUNNING;

CASE _stepClearError OF
  
  0:  // set busy flag
      Busy := TRUE;
      // trigger parameter update to disable FB
     _parameterUpdateInternal := TRUE;
      // call Check Parameter changed method to trigger the parameter update to disable the function
      CheckParameterChanged(AxesGroup := AxesGroup);
      // set timeout
      SetTimeout(PT := _timeoutClearError, rTimer := _timerClearError);
      // inc step counter
     _stepClearError := _stepClearError + 1; 
      
  1: IF ( _responseReceived )
     THEN
       // reset response received flag
      _responseReceived := FALSE;
       // reset step counter
      _stepClearError := 0;
       // finished
       OnExecErrorClear := RobotLibraryConstants.OK;
     ELSE
       // timeout exceeded ? 
       IF (CheckTimeout(_timerClearError) = RobotLibraryConstants.OK)
       THEN
         OnExecErrorClear := RobotLibraryConstants.HAS_ERROR;
       END_IF
	   END_IF
ELSE
  // invalid step
  SetError( ErrorID := RobotLibraryErrorIdEnum.ERR_INVALID_STEP, Overwrite := TRUE );
END_CASE


// reset step counter
IF (OnExecErrorClear <> RobotLibraryConstants.RUNNING)
THEN
  // Reset 
  Reset();     
  // reset step counter
 _stepClearError := 0;
END_IF
                
END_METHOD

METHOD PROTECTED OnExecRun : DINT
VAR_IN_OUT
  /// Robot assignment of function
  AxesGroup : AxesGroup; 
END_VAR
                  // call base implementation
SUPER^.OnExecRun(AxesGroup := AxesGroup);

CASE _stepCmd OF
  
  00:  IF ( _enable_R.Q ) AND ( NOT Error)
       THEN
         // reset the rising edge
        _enable_R();
       
         // Check function is supported and parameter are valid ?
         IF (( CheckFunctionSupported( AxesGroup := AxesGroup )) AND
             ( CheckParameterValid   ( AxesGroup := AxesGroup )))      
         THEN
           // Reset all internal flags
           Reset();
           // set busy flag
           Busy := TRUE;
           // Reset command outputs
           SysDepMemSet(pDest := ADR(OutCmd), Value := 0, DataLen := SIZEOF(OutCmd));         
           // apply command parameter
          _parCmd := ParCmd;
           // init parameter sequence
          _command.ParSeq := 1;
           // create command data
           CommandData := CreateCommandPayload(AxesGroup := AxesGroup);
           // Add command to active command register
          _uniqueID := AxesGroup.Acyclic.ActiveCommandRegister.AddCmd( pCommandFB := ADR(THIS^ ));     
           // set timeout
           SetTimeout(PT := _timeoutCmd, rTimer := _timerCmd);
           // inc step counter
          _stepCmd := _stepCmd + 1; 
         END_IF
       END_IF     


  01:  // Wait for responce received
       IF ( _responseReceived )
       THEN
         // reset response received flag
        _responseReceived := FALSE;
         // update state flags
         OnUpdateStateFlags(_response.State);
         // update state flags
         OnApplyOutCmd(_response.State);
       END_IF
       
       // do not abort directly, so that the ParSeq update can be send
       IF ( _enable_F.Q ) 
       THEN
         // trigger parameter update to disable FB
        _parameterUpdateInternal := TRUE;
         // reset the falling edge
        _enable_F();
         // set timeout
         SetTimeout(PT := _timeoutCmd, rTimer := _timerCmd);
         // inc step counter
        _stepCmd := _stepCmd + 1; 
       END_IF

      // Wait for response received or timeout or not Initialized
  02: IF ((    _responseReceived                                   )  OR 
          (     CheckTimeout(_timerCmd) = RobotLibraryConstants.OK )) OR 
         (( NOT AxesGroup.State.Initialized                        )  AND
          ( NOT AxesGroup.State.Synchronized                       ))
      THEN
        Reset();   
	    END_IF
      
      
ELSE
  // invalid step
  SetError( ErrorID := RobotLibraryErrorIdEnum.ERR_INVALID_STEP, Overwrite := TRUE );
END_CASE



// Reset FB
IF (( _enable_R.Q ) OR
    ( _enable_F.Q ))
THEN
  Reset(); 
END_IF
                
END_METHOD

METHOD PROTECTED OnUpdateStateFlags
VAR_INPUT
  /// Command message state
  State : CmdMessageState;
END_VAR
                  // Reset State flags
;

// Update enable flag
Enabled := _response.Enabled;

CASE State OF

  // No operation or process is active
  CmdMessageState.EMPTY               :;
  // Created but not yet started
  CmdMessageState.CREATED             :;
  // Buffered and awaiting execution
  CmdMessageState.BUFFERED            : CommandBuffered   := TRUE;
                                        ParameterAccepted := TRUE;
  // Buffered in planner for future execution
  CmdMessageState.BUFFERED_IN_PLANNER : CommandBuffered   := TRUE;
                                        ParameterAccepted := TRUE;
  // Currently active and in progress
  CmdMessageState.ACTIVE              : 
  // Interrupted and awaiting continuation
  CmdMessageState.INTERRUPTED         :;
  // Requested for abort
  CmdMessageState.ABORT_REQUEST       :;
  // Successfully completed
  CmdMessageState.DONE                : Busy  := FALSE;
  // Aborted before completion
  CmdMessageState.ABORTED             : Busy  := FALSE;
  // Encountered an error during execution
  CmdMessageState.ERROR               : Error := TRUE;
                                        Busy  := FALSE;
END_CASE
                
END_METHOD

METHOD INTERNAL ParseResponsePayload : DINT
VAR_INPUT
  /// Response data
  ResponseData : RobotLibraryResponseDataFB;
  /// Timestamp
  Timestamp    : SystemTime;  
END_VAR
VAR
  /// Parameter count
 _parameterCnt : DINT;
END_VAR
// Table 6-710: Received CMD payload (RC to PLC) of "AvoidSingularity"
// --------------------------
// Header
// --------------------------
// Byte 00 : USINT - ParSeq | State     
// Byte 01 : SINT  - AlarmMessageSeverity    
// Byte 02 : UINT  - AlarmMessageCode HB
// Byte 03 :       - AlarmMessageCode LB
// --------------------------
// Datablock
// --------------------------
// Byte 04 : BOOL  - Enabled
// --------------------------
                  // call base implementation to parse the header from payload buffer
ResponseData.PayloadPtr := SUPER^.ParseResponsePayload(ResponseData := ResponseData, Timestamp := Timestamp);

// copy parsed header to response
_response.ParSeq               := _rspHeader.ParSeq;
_response.State                := _rspHeader.State;
_response.AlarmMessageSeverity := _rspHeader.AlarmMessageSeverity;
_response.AlarmMessageCode     := _rspHeader.AlarmMessageCode;


// Check payload remaining ? 
IF ( ResponseData.IsPayloadRemaining)
THEN
  // Get Response.Enabled
 _response.Enabled := ResponseData.GetBool();
  // inc parameter counter
 _parameterCnt := _parameterCnt + 1;
END_IF


// Create logging
ParseResponsePayloadLog(ResponseData := ResponseData, Timestamp := Timestamp, ParameterCnt := _parameterCnt);
                
END_METHOD

METHOD INTERNAL ParseResponsePayloadLog
VAR_INPUT
  /// Response data
  ResponseData : RobotLibraryResponseDataFB;
  /// Timestamp
  Timestamp    : SystemTime;  
  /// Parameter count
  ParameterCnt : DINT;
END_VAR
                  // Create log entry for Parameter start
CreateLogMessagePara1 ( Timestamp   := Timestamp,
                        MessageType := MessageType.CMD,
                        Severity    := Severity.DEBUG,
                        MessageCode := 0,
                        MessageText := '{1} parameter(s) to parse from the response data:',
                        Para1       := DINT_TO_STRING(ParameterCnt));
                        

// Return if no parameter is remaining...
IF ( ParameterCnt = 0 ) THEN RETURN; END_IF
// dec remaining parameter(s)                        
ParameterCnt := ParameterCnt - 1;
// Create log entry for Enabled
CreateLogMessagePara1 ( Timestamp   := Timestamp,
                        MessageType := MessageType.CMD,
                        Severity    := Severity.DEBUG,
                        MessageCode := 0,
                        MessageText := 'Response.Enabled = {1}',
                        Para1       :=  BOOL_TO_STRING(_response.Enabled));

                
END_METHOD

METHOD PROTECTED Reset : DINT
VAR_INPUT
END_VAR
                  Reset := SUPER^.Reset();

Busy               := FALSE;
CommandBuffered    := FALSE;


                
END_METHOD
END_FUNCTION_BLOCK

/// Activate robot cycle brake test and give feedback to PLC
FUNCTION_BLOCK MC_BrakeTestFB EXTENDS RobotLibraryBaseExecuteFB
// ------------------------------------------------------------------------- 
//  SRCI Robot Library                                                
// ------------------------------------------------------------------------- 
//                                                                           
//  Object:      BrakeTest                                       
//  Author:      Thorsten Brach                                                
//  Date:        2024-06-01
//
//  Description:                                              
//   
//                                                                           
//  Copyright: 
//    (C) 2024 Thorsten Brach. All rights reserved                                                                                                                                            
//             Licensed under the MIT License.
//                                                                           
//  Disclaimer:                                                                           
//    This project is provided without any guarantee and can be used for   
//    private and commercial purposes. Any use is at the user’s 
//    own risk and responsibility.
//
// -------------------------------------------------------------------------
VAR_INPUT
  /// Command parameter 
  ParCmd             : BrakeTestParCmd;
  /// Parameter which determines the behavior towards the previously sent and still active or buffered commands.
  AbortingMode       : AbortingMode;
  /// Defines the target sequence in which the command will be executed
  SequenceFlag       : SequenceFlag;  
END_VAR
VAR_OUTPUT
  /// Command is transferred and confirmed by the RC
  CommandBuffered    : BOOL;
  /// During the realization of the brake test, the command controls the motion of the respective axis group.
  /// TRUE: The brake test is being realized
  /// FALSE: The brake test is not realized
  Active             : BOOL;
  /// The command was aborted by another command.
  CommandAborted     : BOOL;
  /// TRUE, while command is interrupted during execution and can be continued
  CommandInterrupted : BOOL; 
  /// Command output 
  OutCmd             : BrakeTestOutCmd;
END_VAR

var
  /// internal copy of command parameter 
 _parCmd             : BrakeTestParCmd;
  /// command data to send
 _command            : BrakeTestSendData;
  /// response data received
 _response           : BrakeTestRecvData;      
END_VAR

            SUPER^(AxesGroup := AxesGroup);
          

METHOD INTERNAL CheckAddParameter : BOOL
VAR_INPUT
  /// Payload pointer
  PayloadPtr : UDINT;
END_VAR
VAR
  /// Payload as byte array
  Payload    : ARRAY [1..SIZEOF(_command)] OF BYTE;
  /// Null Byte array 
  Null       : ARRAY [1..SIZEOF(_command)] OF BYTE;
  /// Data length to compare
  DataLen    : UDINT;
END_VAR
                  // Payload pointer must be decreased by one byte, because ADR(Payload) is already one byte !
PayloadPtr := LIMIT (0, PayloadPtr - 1, SIZEOF(Payload) -1);
// Convert command struct to payload array
SysDepMemCpy( pDest := ADR(Payload), pSrc := ADR(_command), DataLen := SIZEOF(_command));
// Calculate the data length to compare - at least one byte must be compared !
DataLen := LIMIT(1, SIZEOF(Payload) - PayloadPtr, SIZEOF(Payload)); 
// Compare Payload-Array with Null-Byte-Array
CheckAddParameter := SysDepMemCmp( pData1 := ADR(Payload) + PayloadPtr , pData2 := ADR(Null), DataLen := DataLen) <>  RobotLibraryConstants.OK ;
                
END_METHOD

METHOD PROTECTED CheckFunctionSupported : BOOL
VAR_IN_OUT
  /// Robot assignment of function
  AxesGroup : AxesGroup; 
END_VAR
                  CheckFunctionSupported := AxesGroup.State.RobotData.RCSupportedFunctions.BrakeTest;

IF ( NOT CheckFunctionSupported )
THEN
  // call base implementation for set error and create log entry
  SUPER^.CheckFunctionSupported(AxesGroup := AxesGroup);
END_IF
                
END_METHOD

METHOD PROTECTED CheckParameterChanged : BOOL
VAR_IN_OUT
  /// Robot assignment of function
  AxesGroup    : AxesGroup; 
END_VAR
                  // Check ParCmd Size is > 0, because MemCmp does not work correctly with size = 0
IF (SIZEOF(ParCmd) = 0) OR (_stepCmd = 0)
THEN 
  RETURN;
END_IF

// compare memory 
_parameterChanged := ( SysDepMemCmp(pData1 := ADR(ParCmd), pData2 := ADR(_parCmd), DataLen := SIZEOF(ParCmd)) <> RobotLibraryConstants.OK );

// check parameter valid ?
_parameterValid   := CheckParameterValid( AxesGroup := AxesGroup );

IF ((  _parameterChanged        )  AND 
    (  _parameterValid          )) OR
    (  _parameterUpdateInternal )  
THEN  
  // Create log entry for parameter changed event
  CreateLogMessagePara1 ( Timestamp   := AxesGroup.State.SystemTime,
                          MessageType := MessageType.CMD,
                          Severity    := Severity.DEBUG,
                          MessageCode := 0,
                          MessageText := 'NotifyParameterChanged Event {1}',
                          Para1       :=  '' );

  // reset internal flag for send parameter update
 _parameterUpdateInternal := FALSE;
  // update internal copy of parameters 
 _parCmd := ParCmd;
  // inc parameter sequence
 _command.ParSeq := _command.ParSeq + 1;
  // update command data  
  CommandData := CreateCommandPayload(AxesGroup := AxesGroup); // ( Access via reference to rCommandFB in ACR )
  // notify active command register 
  AxesGroup.Acyclic.ActiveCommandRegister.NotifyParameterChanged := _uniqueID;  
END_IF
                
END_METHOD

METHOD PROTECTED CheckParameterValid : BOOL
VAR_IN_OUT
  /// Robot assignment of function
  AxesGroup : AxesGroup; 
END_VAR
                  CheckParameterValid := TRUE;

// Check ParCmd.SequenceFlag valid ? 
IF (( SequenceFlag <> SequenceFlagEnum.PRIMARY_SEQUENCE   ) AND  
    ( SequenceFlag <> SequenceFlagEnum.SECONDARY_SEQUENCE ))
THEN
  // Parameter not valid
  CheckParameterValid := FALSE;
  // Set error
  SetError( ErrorID := RobotLibraryErrorIdEnum.ERR_SEQFLAG_NOT_ALLOWED, Overwrite := TRUE );
  // Create log entry
  CreateLogMessagePara1 ( Timestamp   := AxesGroup.State.SystemTime,
                          MessageType := MessageType.CMD,
                          Severity    := Severity.ERROR,
                          MessageCode := ErrorID,
                          MessageText := 'Invalid Parameter SequenceFlag = {1}',
                          Para1       := SEQUENCE_FLAG_TO_STRING (SequenceFlag));
  RETURN;                          
END_IF


// Check AbortingMode valid ? 
IF (( AbortingMode <> AbortingModeEnum.BUFFER ) AND  
    ( AbortingMode <> AbortingModeEnum.ABORT  ))
THEN
  // Parameter not valid
  CheckParameterValid := FALSE;
  // Set error
  SetError( ErrorID := RobotLibraryErrorIdEnum.ERR_ABORTINGMODE_INVALID, Overwrite := TRUE );
  // Create log entry
  CreateLogMessagePara1 ( Timestamp   := AxesGroup.State.SystemTime,
                          MessageType := MessageType.CMD,
                          Severity    := Severity.ERROR,
                          MessageCode := ErrorID,
                          MessageText := 'Invalid Parameter AbortingMode = {1}',
                          Para1       := ABORTING_MODE_TO_STRING(AbortingMode));
  RETURN;                          
END_IF


// Check RobotAxesActive valid ? 
IF ((( ParCmd.RobotAxesActive.AxisJ1 ) AND ( NOT AxesGroup.State.RobotData.AxisJointUsed.J1 )) OR
    (( ParCmd.RobotAxesActive.AxisJ2 ) AND ( NOT AxesGroup.State.RobotData.AxisJointUsed.J2 )) OR
    (( ParCmd.RobotAxesActive.AxisJ3 ) AND ( NOT AxesGroup.State.RobotData.AxisJointUsed.J3 )) OR
    (( ParCmd.RobotAxesActive.AxisJ4 ) AND ( NOT AxesGroup.State.RobotData.AxisJointUsed.J4 )) OR
    (( ParCmd.RobotAxesActive.AxisJ5 ) AND ( NOT AxesGroup.State.RobotData.AxisJointUsed.J5 )) OR
    (( ParCmd.RobotAxesActive.AxisJ6 ) AND ( NOT AxesGroup.State.RobotData.AxisJointUsed.J6 )))  
THEN
  // Parameter not valid
  CheckParameterValid := FALSE;
  // Set error
  SetError( ErrorID := RobotLibraryErrorIdEnum.ERR_INVALID_PAR_CMD, Overwrite := TRUE );
  // Create log entry
  CreateLogMessagePara1 ( Timestamp   := AxesGroup.State.SystemTime,
                          MessageType := MessageType.CMD,
                          Severity    := Severity.ERROR,
                          MessageCode := ErrorID,
                          MessageText := 'Invalid Parameter ParCmd.RobotAxesActive = {1}',
                          Para1       := ROBOT_AXES_FLAGS_TO_STRING(ParCmd.RobotAxesActive));
  RETURN;                          
END_IF


// Check ExternalAxesActive valid ? 
IF ((( ParCmd.ExternalAxesActive.AxisE1 ) AND ( NOT AxesGroup.State.RobotData.AxisExternalUsed.E1 )) OR
    (( ParCmd.ExternalAxesActive.AxisE2 ) AND ( NOT AxesGroup.State.RobotData.AxisExternalUsed.E2 )) OR
    (( ParCmd.ExternalAxesActive.AxisE3 ) AND ( NOT AxesGroup.State.RobotData.AxisExternalUsed.E3 )) OR
    (( ParCmd.ExternalAxesActive.AxisE4 ) AND ( NOT AxesGroup.State.RobotData.AxisExternalUsed.E4 )) OR
    (( ParCmd.ExternalAxesActive.AxisE5 ) AND ( NOT AxesGroup.State.RobotData.AxisExternalUsed.E5 )) OR
    (( ParCmd.ExternalAxesActive.AxisE6 ) AND ( NOT AxesGroup.State.RobotData.AxisExternalUsed.E6 )))  
THEN
  // Parameter not valid
  CheckParameterValid := FALSE;
  // Set error
  SetError( ErrorID := RobotLibraryErrorIdEnum.ERR_INVALID_PAR_CMD, Overwrite := TRUE );
  // Create log entry
  CreateLogMessagePara1 ( Timestamp   := AxesGroup.State.SystemTime,
                          MessageType := MessageType.CMD,
                          Severity    := Severity.ERROR,
                          MessageCode := ErrorID,
                          MessageText := 'Invalid Parameter ParCmd.ExternalAxesActive = {1}',
                          Para1       := EXTERNAL_AXES_FLAGS_TO_STRING(ParCmd.ExternalAxesActive));
  RETURN;                          
END_IF
                
END_METHOD

METHOD INTERNAL CreateCommandPayload : RobotLibraryCommandDataFB
VAR_IN_OUT
  /// Robot assignment of function
  AxesGroup : AxesGroup; 
END_VAR
VAR
  /// Parameter count
 _parameterCnt : DINT;
END_VAR
// Table 6-740: Sent CMD payload (PLC to RC) of "BrakeTest"
// --------------------------
// Header
// --------------------------
// Byte 00 : UINT  - Type HB     
// Byte 01 :       - Type LB    
// Byte 02 : USINT - Reserve | ExecutionMode
// Byte 03 : USINT - ParSeq  | Priority
// --------------------------
// Datablock
// --------------------------
// Byte 04 : BYTE - RobotAxesActive
// Byte 05 : BYTE - ExternalAxesActive
// --------------------------
                  // set command parameter 
_command.CmdTyp               :=  CmdType.BrakeTest;
_command.ExecMode             :=  ExecMode;
_command.ParSeq               := _command.ParSeq;
_command.Priority             :=  Priority;
_command.RobotAxesActive.0    := _parCmd.RobotAxesActive.Bit00;
_command.RobotAxesActive.1    := _parCmd.RobotAxesActive.AxisJ1;
_command.RobotAxesActive.2    := _parCmd.RobotAxesActive.AxisJ2;
_command.RobotAxesActive.3    := _parCmd.RobotAxesActive.AxisJ3;
_command.RobotAxesActive.4    := _parCmd.RobotAxesActive.AxisJ4;
_command.RobotAxesActive.5    := _parCmd.RobotAxesActive.AxisJ5;
_command.RobotAxesActive.6    := _parCmd.RobotAxesActive.AxisJ6;
_command.RobotAxesActive.7    := _parCmd.RobotAxesActive.Bit07;
_command.ExternalAxesActive.0 := _parCmd.ExternalAxesActive.Bit00;
_command.ExternalAxesActive.1 := _parCmd.ExternalAxesActive.AxisE1;
_command.ExternalAxesActive.2 := _parCmd.ExternalAxesActive.AxisE2;
_command.ExternalAxesActive.3 := _parCmd.ExternalAxesActive.AxisE3;
_command.ExternalAxesActive.4 := _parCmd.ExternalAxesActive.AxisE4;
_command.ExternalAxesActive.5 := _parCmd.ExternalAxesActive.AxisE5;
_command.ExternalAxesActive.6 := _parCmd.ExternalAxesActive.AxisE6;
_command.ExternalAxesActive.7 := _parCmd.ExternalAxesActive.Bit07;

// copy command data to header
_cmdHeader := _command;
// call base implementation to copy header to payload buffer
CreateCommandPayload := SUPER^.CreateCommandPayload(AxesGroup := AxesGroup);


// Check parameter must be added ? 
IF ( CheckAddParameter(CreateCommandPayload.PayloadPtr))
THEN
  // add command.EmitterID[0]
  CreateCommandPayload.AddByte(_command.RobotAxesActive);
  // inc parameter counter
 _parameterCnt := _parameterCnt + 1;  
END_IF


// Check parameter must be added ? 
IF ( CheckAddParameter(CreateCommandPayload.PayloadPtr))
THEN
  // add command.EmitterID[1]
  CreateCommandPayload.AddByte(_command.ExternalAxesActive);
  // inc parameter counter
 _parameterCnt := _parameterCnt + 1;  
END_IF


// Create logging
CreateCommandPayloadLog(AxesGroup := AxesGroup, ParameterCnt := _parameterCnt);
                
END_METHOD

METHOD INTERNAL CreateCommandPayloadLog
VAR_IN_OUT
  /// Robot assignment of function
  AxesGroup : AxesGroup; 
END_VAR
VAR_INPUT
  /// Parameter count
  ParameterCnt : DINT;
END_VAR
                  // Create log entry for Parameter start
CreateLogMessagePara1 ( Timestamp   := AxesGroup.State.SystemTime,
                        MessageType := MessageType.CMD,
                        Severity    := Severity.DEBUG,
                        MessageCode := 0,
                        MessageText := 'Create command payload with {1} parameter(s) :',
                        Para1       := DINT_TO_STRING(ParameterCnt));
  

// Return if no parameter is remaining...
IF ( ParameterCnt = 0 ) THEN RETURN; END_IF
// dec remaining parameter(s)                        
ParameterCnt := ParameterCnt - 1;
// Create log entry for RobotAxesActive
CreateLogMessagePara1 ( Timestamp   := AxesGroup.State.SystemTime,
                        MessageType := MessageType.CMD,
                        Severity    := Severity.DEBUG,
                        MessageCode := 0,
                        MessageText := 'Command.RobotAxesActive = {1}',
                        Para1       :=  BYTE_TO_STRING_BIN(_command.RobotAxesActive));


// Return if no parameter is remaining...
IF ( ParameterCnt = 0 ) THEN RETURN; END_IF
// dec remaining parameter(s)                        
ParameterCnt := ParameterCnt - 1;
// Create log entry for ExternalAxesActive
CreateLogMessagePara1 ( Timestamp   := AxesGroup.State.SystemTime,
                        MessageType := MessageType.CMD,
                        Severity    := Severity.DEBUG,
                        MessageCode := 0,
                        MessageText := 'Command.ExternalAxesActive = {1}',
                        Para1       :=  BYTE_TO_STRING_BIN(_command.ExternalAxesActive));


                
END_METHOD

METHOD FB_init : BOOL
VAR_INPUT
  /// if TRUE, the retain variables are initialized (warm start / cold start)
  bInitRetains : BOOL; 
  /// if TRUE, the instance afterwards gets moved into the copy code (online change)
  bInCopyCode  : BOOL;  
END_VAR
                  MyType := 'MC_BrakeTestFB';

ExecMode     := ExecutionMode.SEQUENCE_PRIMARY;
Priority     := PriorityLevel.NORMAL;
SequenceFlag := SequenceFlagEnum.PRIMARY_SEQUENCE;  

                
END_METHOD

METHOD PROTECTED OnApplyOutCmd
VAR_INPUT
  /// Command message state
  State : CmdMessageState;
END_VAR
                  IF ( State = CmdMessageState.EMPTY ) 
THEN
  // Reset command outputs
  SysDepMemSet(pDest := ADR(OutCmd), Value := 0, DataLen := SIZEOF(OutCmd));         
END_IF

IF ( State = CmdMessageState.DONE )
THEN
  // Update results
  OutCmd.RobotAxesStatus.Bit00     := _response.RobotAxesStatus.0;
  OutCmd.RobotAxesStatus.AxisJ1    := _response.RobotAxesStatus.1;
  OutCmd.RobotAxesStatus.AxisJ2    := _response.RobotAxesStatus.2;
  OutCmd.RobotAxesStatus.AxisJ3    := _response.RobotAxesStatus.3;
  OutCmd.RobotAxesStatus.AxisJ4    := _response.RobotAxesStatus.4;
  OutCmd.RobotAxesStatus.AxisJ5    := _response.RobotAxesStatus.5;
  OutCmd.RobotAxesStatus.AxisJ6    := _response.RobotAxesStatus.6;
  OutCmd.RobotAxesStatus.Bit07     := _response.RobotAxesStatus.7;
  
  OutCmd.RobotAxesWarning.Bit00     := _response.RobotAxesWarning.0;
  OutCmd.RobotAxesWarning.AxisJ1    := _response.RobotAxesWarning.1;
  OutCmd.RobotAxesWarning.AxisJ2    := _response.RobotAxesWarning.2;
  OutCmd.RobotAxesWarning.AxisJ3    := _response.RobotAxesWarning.3;
  OutCmd.RobotAxesWarning.AxisJ4    := _response.RobotAxesWarning.4;
  OutCmd.RobotAxesWarning.AxisJ5    := _response.RobotAxesWarning.5;
  OutCmd.RobotAxesWarning.AxisJ6    := _response.RobotAxesWarning.6;
  OutCmd.RobotAxesWarning.Bit07     := _response.RobotAxesWarning.7;
  
  OutCmd.ExternalAxesStatus.Bit00   := _response.ExternalAxesStatus.0;
  OutCmd.ExternalAxesStatus.AxisE1  := _response.ExternalAxesStatus.1;
  OutCmd.ExternalAxesStatus.AxisE2  := _response.ExternalAxesStatus.2;
  OutCmd.ExternalAxesStatus.AxisE3  := _response.ExternalAxesStatus.3;
  OutCmd.ExternalAxesStatus.AxisE4  := _response.ExternalAxesStatus.4;
  OutCmd.ExternalAxesStatus.AxisE5  := _response.ExternalAxesStatus.5;
  OutCmd.ExternalAxesStatus.AxisE6  := _response.ExternalAxesStatus.6;
  OutCmd.ExternalAxesStatus.Bit07   := _response.ExternalAxesStatus.7;
  
  OutCmd.ExternalAxesWarning.Bit00  := _response.ExternalAxesWarning.0;
  OutCmd.ExternalAxesWarning.AxisE1 := _response.ExternalAxesWarning.1;
  OutCmd.ExternalAxesWarning.AxisE2 := _response.ExternalAxesWarning.2;
  OutCmd.ExternalAxesWarning.AxisE3 := _response.ExternalAxesWarning.3;
  OutCmd.ExternalAxesWarning.AxisE4 := _response.ExternalAxesWarning.4;
  OutCmd.ExternalAxesWarning.AxisE5 := _response.ExternalAxesWarning.5;
  OutCmd.ExternalAxesWarning.AxisE6 := _response.ExternalAxesWarning.6;
  OutCmd.ExternalAxesWarning.Bit07  := _response.ExternalAxesWarning.7;
END_IF
                
END_METHOD

METHOD PROTECTED OnExecRun : DINT
VAR_IN_OUT
  /// Robot assignment of function
  AxesGroup : AxesGroup; 
END_VAR
                  // call base implementation
SUPER^.OnExecRun(AxesGroup := AxesGroup);

CASE _stepCmd OF
  
  00:  IF ( _execute_R.Q ) AND ( NOT Error) 
       THEN
         // Check function is supported and parameter are valid ?
         IF (( CheckFunctionSupported( AxesGroup := AxesGroup )) AND
             ( CheckParameterValid   ( AxesGroup := AxesGroup )))      
         THEN
           // set busy flag
           Busy := TRUE;
           // Reset command outputs
           SysDepMemSet(pDest := ADR(OutCmd), Value := 0, DataLen := SIZEOF(OutCmd));         
           // apply command parameter
          _parCmd := ParCmd;
           // init parameter sequence
          _command.ParSeq := 1;
           // create command data
           CommandData := CreateCommandPayload(AxesGroup := AxesGroup);
           // Add command to active command register
          _uniqueID := AxesGroup.Acyclic.ActiveCommandRegister.AddCmd( pCommandFB := ADR(THIS^ ));     
           // set timeout
           SetTimeout(PT := _timeoutCmd, rTimer := _timerCmd);
           // inc step counter
          _stepCmd := _stepCmd + 1;
         END_IF 
       END_IF
     

  01:  // Wait for responce received
       IF ( _responseReceived )
       THEN
         // reset response received flag
        _responseReceived := FALSE;
         // update state flags
         OnUpdateStateFlags(_response.State);
         // update state flags
         OnApplyOutCmd(_response.State);
                
         // Done, Aborted or Error ?
         IF (_response.State >= CmdMessageState.DONE )
         THEN 
           // set timeout
           SetTimeout(PT := _timeoutCmd, rTimer := _timerCmd);
           // inc step counter
          _stepCmd := _stepCmd + 1; 
         END_IF
       END_IF

  02: IF ( NOT Execute)
      THEN
        Reset();
      END_IF     
ELSE
  // invalid step
  SetError( ErrorID := RobotLibraryErrorIdEnum.ERR_INVALID_STEP, Overwrite := TRUE );
END_CASE


// Reset FB
IF ( NOT Execute )
THEN
  Reset();  
END_IF
                
END_METHOD

METHOD PROTECTED OnUpdateStateFlags
VAR_INPUT
  /// Command message state
  State : CmdMessageState;
END_VAR
                  // Reset State flags
Active             := FALSE;
CommandAborted     := FALSE;
CommandInterrupted := FALSE;
Done               := FALSE;

CASE State OF

  // No operation or process is active
  CmdMessageState.EMPTY               :;
  // Created but not yet started
  CmdMessageState.CREATED             :;
  // Buffered and awaiting execution
  CmdMessageState.BUFFERED            : CommandBuffered    := TRUE;
  // Buffered in planner for future execution
  CmdMessageState.BUFFERED_IN_PLANNER : CommandBuffered    := TRUE;
  // Currently active and in progress
  CmdMessageState.ACTIVE              : Active             := TRUE;
  // Interrupted and awaiting continuation
  CmdMessageState.INTERRUPTED         : CommandInterrupted := TRUE;
  // Requested for abort
  CmdMessageState.ABORT_REQUEST       :;
  // Successfully completed
  CmdMessageState.DONE                : Done               := TRUE;
                                        Busy               := FALSE;
  // Aborted before completion
  CmdMessageState.ABORTED             : CommandAborted     := TRUE;
                                        Busy               := FALSE;
  // Encountered an error during execution
  CmdMessageState.ERROR               : Error              := TRUE;
                                        Busy               := FALSE;
END_CASE
                
END_METHOD

METHOD INTERNAL ParseResponsePayload : DINT
VAR_INPUT
  /// Response data
  ResponseData : RobotLibraryResponseDataFB;
  /// Timestamp
  Timestamp    : SystemTime;  
END_VAR
VAR
  /// Parameter count
 _parameterCnt : DINT;
END_VAR
// Table 6-741: Received CMD payload (RC to PLC) of "BrakeTest"
// --------------------------
// Header
// --------------------------
// Byte 00 : USINT - ParSeq | State     
// Byte 01 : SINT  - AlarmMessageSeverity    
// Byte 02 : UINT  - AlarmMessageCode HB
// Byte 03 :       - AlarmMessageCode LB
// --------------------------
// Datablock
// --------------------------
// Byte 04 : BYTE  - RobotAxesStatus
// Byte 05 : BYTE  - ExternalAxesStatus
// Byte 06 : BYTE  - RobotAxesWarning
// Byte 07 : BYTE  - ExternalAxesWarning
// --------------------------
                  // call base implementation to parse the header from payload buffer
ResponseData.PayloadPtr := SUPER^.ParseResponsePayload(ResponseData := ResponseData, Timestamp := Timestamp);

// copy parsed header to response
_response.ParSeq               := _rspHeader.ParSeq;
_response.State                := _rspHeader.State;
_response.AlarmMessageSeverity := _rspHeader.AlarmMessageSeverity;
_response.AlarmMessageCode     := _rspHeader.AlarmMessageCode;

// Check payload remaining ? 
IF ( ResponseData.IsPayloadRemaining)
THEN
  // Get RobotAxesStatus
 _response.RobotAxesStatus := ResponseData.GetByte();
  // inc parameter counter
 _parameterCnt := _parameterCnt + 1;
END_IF


// Check payload remaining ? 
IF ( ResponseData.IsPayloadRemaining)
THEN
  // Get ExternalAxesStatus
 _response.ExternalAxesStatus := ResponseData.GetByte();
  // inc parameter counter
 _parameterCnt := _parameterCnt + 1;
END_IF


// Check payload remaining ? 
IF ( ResponseData.IsPayloadRemaining)
THEN
  // Get RobotAxesWarning
 _response.RobotAxesWarning := ResponseData.GetByte();
  // inc parameter counter
 _parameterCnt := _parameterCnt + 1;
END_IF


// Check payload remaining ? 
IF ( ResponseData.IsPayloadRemaining)
THEN
  // Get ExternalAxesWarning
 _response.ExternalAxesWarning := ResponseData.GetByte();
  // inc parameter counter
 _parameterCnt := _parameterCnt + 1;
END_IF


// Create logging
ParseResponsePayloadLog(ResponseData := ResponseData, Timestamp := Timestamp, ParameterCnt := _parameterCnt);
                
END_METHOD

METHOD INTERNAL ParseResponsePayloadLog
VAR_INPUT
  /// Response data
  ResponseData : RobotLibraryResponseDataFB;
  /// Timestamp
  Timestamp    : SystemTime;  
  /// Parameter count
  ParameterCnt : DINT;
END_VAR
                  // Create log entry for Parameter start
CreateLogMessagePara1 ( Timestamp   := Timestamp,
                        MessageType := MessageType.CMD,
                        Severity    := Severity.DEBUG,
                        MessageCode := 0,
                        MessageText := '{1} parameter(s) to parse from the response data:',
                        Para1       := DINT_TO_STRING(ParameterCnt));


// Return if no parameter is remaining...
IF ( ParameterCnt = 0 ) THEN RETURN; END_IF
// dec remaining parameter(s)                        
ParameterCnt := ParameterCnt - 1;
// Create log entry for RobotAxesStatus
CreateLogMessagePara1 ( Timestamp   := Timestamp,
                        MessageType := MessageType.CMD,
                        Severity    := Severity.DEBUG,
                        MessageCode := 0,
                        MessageText := 'Response.RobotAxesStatus = {1}',
                        Para1       :=  BYTE_TO_STRING_BIN(_response.RobotAxesStatus));


// Return if no parameter is remaining...
IF ( ParameterCnt = 0 ) THEN RETURN; END_IF
// dec remaining parameter(s)                        
ParameterCnt := ParameterCnt - 1;
// Create log entry for ExternalAxesStatus
CreateLogMessagePara1 ( Timestamp   := Timestamp,
                        MessageType := MessageType.CMD,
                        Severity    := Severity.DEBUG,
                        MessageCode := 0,
                        MessageText := 'Response.ExternalAxesStatus = {1}',
                        Para1       :=  BYTE_TO_STRING_BIN(_response.ExternalAxesStatus));


// Return if no parameter is remaining...
IF ( ParameterCnt = 0 ) THEN RETURN; END_IF
// dec remaining parameter(s)                        
ParameterCnt := ParameterCnt - 1;
// Create log entry for RobotAxesWarning
CreateLogMessagePara1 ( Timestamp   := Timestamp,
                        MessageType := MessageType.CMD,
                        Severity    := Severity.DEBUG,
                        MessageCode := 0,
                        MessageText := 'Response.RobotAxesWarning = {1}',
                        Para1       :=  BYTE_TO_STRING_BIN(_response.RobotAxesWarning));


// Return if no parameter is remaining...
IF ( ParameterCnt = 0 ) THEN RETURN; END_IF
// dec remaining parameter(s)                        
ParameterCnt := ParameterCnt - 1;
// Create log entry for ExternalAxesWarning
CreateLogMessagePara1 ( Timestamp   := Timestamp,
                        MessageType := MessageType.CMD,
                        Severity    := Severity.DEBUG,
                        MessageCode := 0,
                        MessageText := 'Response.ExternalAxesWarning = {1}',
                        Para1       :=  BYTE_TO_STRING_BIN(_response.ExternalAxesWarning));
                
END_METHOD

METHOD PROTECTED Reset : DINT
VAR_INPUT
END_VAR
                  Reset := SUPER^.Reset();

Done               := FALSE;
Busy               := FALSE;
Active             := FALSE;
CommandBuffered    := FALSE;
CommandAborted     := FALSE;
CommandInterrupted := FALSE; 

                
END_METHOD
END_FUNCTION_BLOCK

/// Call subprogram stored in RC from PLC
FUNCTION_BLOCK MC_CallSubprogramFB EXTENDS RobotLibraryBaseExecuteFB
// ------------------------------------------------------------------------- 
//  SRCI Robot Library                                                
// ------------------------------------------------------------------------- 
//                                                                           
//  Object:      CallSubprogramFB                                       
//  Author:      Thorsten Brach                                                
//  Date:        2024-06-01
//
//  Description:                                              
//   
//                                                                           
//  Copyright: 
//    (C) 2024 Thorsten Brach. All rights reserved                                                                                                                                            
//             Licensed under the MIT License.
//                                                                           
//  Disclaimer:                                                                           
//    This project is provided without any guarantee and can be used for   
//    private and commercial purposes. Any use is at the user’s 
//    own risk and responsibility.
//
// -------------------------------------------------------------------------
VAR_INPUT
  /// command parameter 
  ParCmd             : CallSubprogramParCmd;
  /// Processing mode
  ProcessingMode     : ProcessingMode;
  /// Defines the target sequence in which the command will be executed
  SequenceFlag       : SequenceFlag;
END_VAR

VAR_OUTPUT
  /// TRUE while the output ReturnData returns valid data according to the user defined subprogram
  Valid              : BOOL;
  /// Command is transferred and confirmed by the RC
  CommandBuffered    : BOOL;
  /// The requested subprogram on the RC is in progress. Movement of the axes trough this subprogram is possible.  
  InProgress         : BOOL;
  /// The command was aborted by another command
  CommandAborted     : BOOL;
  /// TRUE, while command is interrupted during execution and can be continued.
  CommandInterrupted : BOOL;
  /// Receiving of input parameter values has been acknowledged by RC
  ParameterAccepted  : BOOL;
  /// command outputs
  OutCmd             : CallSubprogramOutCmd;       
END_VAR



VAR
  /// internal copy of command parameter 
 _parCmd             : CallSubprogramParCmd;
  /// command data to send
 _command            : CallSubprogramSendData;
  /// response data received
 _response           : CallSubprogramRecvData;      
END_VAR

            SUPER^(AxesGroup := AxesGroup);
          

METHOD INTERNAL CheckAddParameter : BOOL
VAR_INPUT
  /// Payload pointer
  PayloadPtr : UDINT;
END_VAR
VAR
  /// Payload as byte array
  Payload    : ARRAY [1..SIZEOF(_command)] OF BYTE;
  /// Null Byte array 
  Null       : ARRAY [1..SIZEOF(_command)] OF BYTE;
  /// Data length to compare
  DataLen    : UDINT;
END_VAR
                  // Payload pointer must be decreased by one byte, because ADR(Payload) is already one byte !
PayloadPtr := LIMIT (0, PayloadPtr - 1, SIZEOF(Payload) -1);
// Convert command struct to payload array
SysDepMemCpy( pDest := ADR(Payload), pSrc := ADR(_command), DataLen := SIZEOF(_command));
// Calculate the data length to compare - at least one byte must be compared !
DataLen := LIMIT(1, SIZEOF(Payload) - PayloadPtr, SIZEOF(Payload)); 
// Compare Payload-Array with Null-Byte-Array
CheckAddParameter := SysDepMemCmp( pData1 := ADR(Payload) + PayloadPtr , pData2 := ADR(Null), DataLen := DataLen) <>  RobotLibraryConstants.OK ;
                
END_METHOD

METHOD PROTECTED CheckFunctionSupported : BOOL
VAR_IN_OUT
  /// Robot assignment of function
  AxesGroup : AxesGroup; 
END_VAR
                  CheckFunctionSupported := AxesGroup.State.RobotData.RCSupportedFunctions.CallSubprogram;

IF ( NOT CheckFunctionSupported )
THEN
  // call base implementation for set error and create log entry
  SUPER^.CheckFunctionSupported(AxesGroup := AxesGroup);
END_IF
                
END_METHOD

METHOD PROTECTED CheckParameterChanged : BOOL
VAR_IN_OUT
  /// Robot assignment of function
  AxesGroup    : AxesGroup; 
END_VAR
                  // Check ParCmd Size is > 0, because MemCmp does not work correctly with size = 0
IF (SIZEOF(ParCmd) = 0) OR (_stepCmd = 0)
THEN 
  RETURN;
END_IF

// compare memory 
_parameterChanged := ( SysDepMemCmp(pData1 := ADR(ParCmd), pData2 := ADR(_parCmd), DataLen := SIZEOF(ParCmd)) <> RobotLibraryConstants.OK );

// check parameter valid ?
_parameterValid   := CheckParameterValid( AxesGroup := AxesGroup );

IF ((  _parameterChanged        )  AND 
    (  _parameterValid          )) OR
    (  _parameterUpdateInternal )  
THEN  
  // Create log entry for parameter changed event
  CreateLogMessagePara1 ( Timestamp   := AxesGroup.State.SystemTime,
                          MessageType := MessageType.CMD,
                          Severity    := Severity.DEBUG,
                          MessageCode := 0,
                          MessageText := 'NotifyParameterChanged Event {1}',
                          Para1       :=  '' );

  // reset internal flag for send parameter update
 _parameterUpdateInternal := FALSE;
  // update internal copy of parameters 
 _parCmd := ParCmd;
  // inc parameter sequence
 _command.ParSeq := _command.ParSeq + 1;
  // update command data  
  CommandData := CreateCommandPayload(AxesGroup := AxesGroup); // ( Access via reference to rCommandFB in ACR )
  // notify active command register 
  AxesGroup.Acyclic.ActiveCommandRegister.NotifyParameterChanged := _uniqueID;  
  // Reset Valid output of the FB 
  Valid := FALSE;
  // Reset parameter accepted flag
  ParameterAccepted := FALSE;
END_IF
                
END_METHOD

METHOD PROTECTED CheckParameterValid : BOOL
VAR_IN_OUT
  /// Robot assignment of function
  AxesGroup : AxesGroup; 
END_VAR

VAR
  /// internal index for loops
 _idx : DINT;
END_VAR
                  CheckParameterValid := TRUE;

